Yaskawa INFORM job: A_ROOF_UPPER_0614_2_PAINT_62.JBI

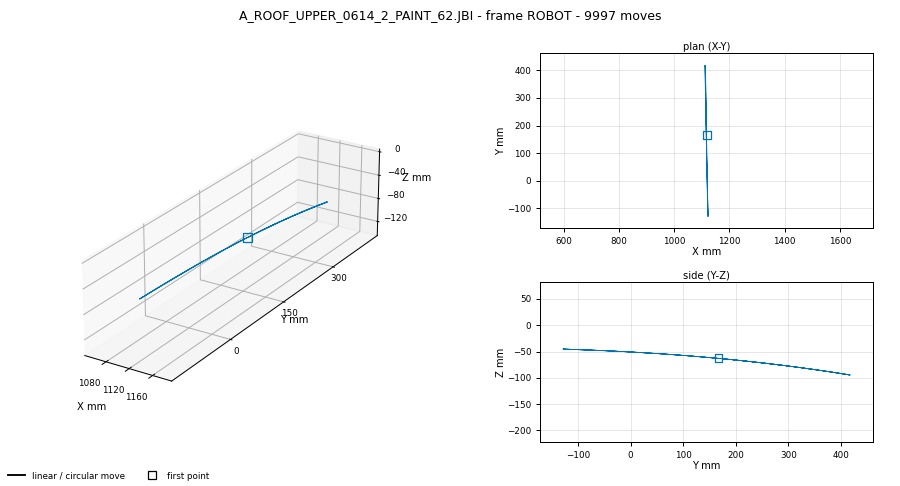
[picture p0: tool path of A_ROOF_UPPER_0614_2_PAINT_62.JBI in frame ROBOT, 9997 of 9997 moves have a stored position in this frame; points joined in program order, loops and branches not executed]
/JOB
//NAME A_ROOF_UPPER_0614_2_PAINT62
//POS
///NPOS 9997,0,0,0,0,0
///TOOL 1
///USER 0
///POSTYPE ROBOT
///RECTAN
///RCONF 1,0,0,0,0,0,0,0,0,0,0,0,0,0,0,0,0,0,0,0,0,0,0,0
C00000=1117.726,167.030,-62.893,-179.337,8.959,149.560
C00001=1117.722,167.279,-62.915,-179.335,8.962,149.560
C00002=1117.717,167.528,-62.939,-179.333,8.966,149.560
C00003=1117.713,167.777,-62.962,-179.330,8.969,149.560
C00004=1117.708,168.025,-62.984,-179.328,8.972,149.560
C00005=1117.703,168.274,-63.008,-179.326,8.975,149.560
C00006=1117.699,168.523,-63.031,-179.324,8.978,149.560
C00007=1117.695,168.772,-63.054,-179.321,8.981,149.560
C00008=1117.690,169.021,-63.077,-179.319,8.985,149.561
C00009=1117.685,169.270,-63.101,-179.317,8.988,149.561
C00010=1117.681,169.519,-63.124,-179.315,8.990,149.561
C00011=1117.676,169.767,-63.146,-179.313,8.993,149.561
C00012=1117.671,170.016,-63.170,-179.310,8.997,149.561
C00013=1117.667,170.265,-63.193,-179.308,9.000,149.561
C00014=1117.662,170.514,-63.217,-179.306,9.002,149.561
C00015=1117.658,170.763,-63.239,-179.304,9.005,149.561
C00016=1117.653,170.977,-63.260,-179.302,9.008,149.561
C00017=1117.650,171.190,-63.279,-179.300,9.010,149.561
C00018=1117.646,171.404,-63.299,-179.298,9.014,149.562
C00019=1117.642,171.619,-63.319,-179.296,9.016,149.562
C00020=1117.638,171.833,-63.339,-179.294,9.018,149.562
C00021=1117.634,172.046,-63.359,-179.292,9.021,149.562
C00022=1117.630,172.260,-63.379,-179.291,9.023,149.562
C00023=1117.626,172.474,-63.399,-179.288,9.026,149.562
C00024=1117.621,172.723,-63.422,-179.286,9.029,149.562
C00025=1117.617,172.971,-63.446,-179.284,9.032,149.562
C00026=1117.613,173.220,-63.469,-179.282,9.035,149.562
C00027=1117.608,173.469,-63.493,-179.280,9.038,149.562
C00028=1117.603,173.718,-63.516,-179.278,9.041,149.562
C00029=1117.599,173.967,-63.539,-179.275,9.044,149.562
C00030=1117.594,174.216,-63.563,-179.273,9.047,149.563
C00031=1117.590,174.464,-63.587,-179.271,9.050,149.563
C00032=1117.585,174.713,-63.610,-179.269,9.053,149.563
C00033=1117.581,174.962,-63.633,-179.267,9.056,149.563
C00034=1117.576,175.211,-63.656,-179.264,9.059,149.563
C00035=1117.572,175.460,-63.680,-179.262,9.062,149.563
C00036=1117.567,175.709,-63.704,-179.260,9.064,149.563
C00037=1117.562,175.958,-63.727,-179.258,9.068,149.563
C00038=1117.558,176.207,-63.750,-179.256,9.071,149.563
C00039=1117.553,176.455,-63.775,-179.254,9.073,149.563
C00040=1117.549,176.704,-63.798,-179.251,9.076,149.564
C00041=1117.544,176.953,-63.821,-179.249,9.080,149.564
C00042=1117.540,177.202,-63.845,-179.247,9.082,149.564
C00043=1117.535,177.451,-63.869,-179.245,9.085,149.564
C00044=1117.530,177.700,-63.892,-179.242,9.089,149.564
C00045=1117.526,177.948,-63.916,-179.241,9.091,149.564
C00046=1117.521,178.197,-63.939,-179.238,9.094,149.564
C00047=1117.517,178.445,-63.964,-179.236,9.098,149.564
C00048=1117.512,178.694,-63.987,-179.234,9.100,149.564
C00049=1117.507,178.943,-64.010,-179.232,9.103,149.564
C00050=1117.503,179.192,-64.034,-179.230,9.106,149.565
C00051=1117.499,179.442,-64.058,-179.228,9.109,149.565
C00052=1117.494,179.690,-64.082,-179.224,9.113,149.565
C00053=1117.490,179.939,-64.106,-179.222,9.116,149.565
C00054=1117.485,180.187,-64.130,-179.219,9.119,149.565
C00055=1117.481,180.437,-64.153,-179.217,9.122,149.565
C00056=1117.476,180.685,-64.177,-179.214,9.125,149.565
C00057=1117.471,180.934,-64.200,-179.211,9.128,149.565
C00058=1117.467,181.182,-64.224,-179.209,9.131,149.565
C00059=1117.462,181.432,-64.248,-179.206,9.134,149.565
C00060=1117.458,181.681,-64.273,-179.204,9.137,149.565
C00061=1117.453,181.930,-64.296,-179.201,9.141,149.565
C00062=1117.449,182.178,-64.320,-179.199,9.144,149.565
C00063=1117.444,182.427,-64.344,-179.196,9.147,149.565
C00064=1117.440,182.676,-64.368,-179.194,9.150,149.565
C00065=1117.435,182.924,-64.392,-179.191,9.153,149.565
C00066=1117.430,183.173,-64.416,-179.189,9.156,149.565
C00067=1117.426,183.423,-64.440,-179.186,9.159,149.565
C00068=1117.422,183.671,-64.464,-179.183,9.162,149.565
C00069=1117.417,183.920,-64.488,-179.181,9.165,149.565
C00070=1117.413,184.168,-64.512,-179.178,9.168,149.565
C00071=1117.407,184.417,-64.536,-179.176,9.171,149.565
C00072=1117.404,184.631,-64.557,-179.174,9.174,149.565
C00073=1117.400,184.845,-64.578,-179.172,9.176,149.565
C00074=1117.396,185.059,-64.598,-179.170,9.178,149.565
C00075=1117.393,185.272,-64.619,-179.167,9.181,149.565
C00076=1117.388,185.485,-64.640,-179.166,9.184,149.565
C00077=1117.384,185.699,-64.660,-179.164,9.186,149.565
C00078=1117.381,185.913,-64.681,-179.162,9.188,149.565
C00079=1117.377,186.127,-64.702,-179.159,9.191,149.566
C00080=1117.372,186.375,-64.726,-179.157,9.194,149.566
C00081=1117.368,186.624,-64.750,-179.154,9.197,149.565
C00082=1117.363,186.873,-64.775,-179.152,9.200,149.565
C00083=1117.359,187.122,-64.799,-179.150,9.202,149.565
C00084=1117.354,187.371,-64.822,-179.147,9.205,149.566
C00085=1117.350,187.620,-64.847,-179.145,9.208,149.566
C00086=1117.345,187.868,-64.871,-179.143,9.211,149.566
C00087=1117.341,188.117,-64.896,-179.140,9.214,149.566
C00088=1117.336,188.366,-64.920,-179.138,9.217,149.566
C00089=1117.332,188.615,-64.945,-179.136,9.219,149.566
C00090=1117.327,188.863,-64.969,-179.134,9.222,149.566
C00091=1117.322,189.112,-64.993,-179.131,9.225,149.566
C00092=1117.318,189.360,-65.017,-179.129,9.228,149.566
C00093=1117.313,189.610,-65.042,-179.127,9.231,149.566
C00094=1117.309,189.858,-65.067,-179.125,9.233,149.566
C00095=1117.305,190.106,-65.091,-179.122,9.236,149.566
C00096=1117.300,190.356,-65.115,-179.120,9.239,149.566
C00097=1117.295,190.605,-65.139,-179.118,9.242,149.566
C00098=1117.291,190.853,-65.164,-179.116,9.244,149.566
C00099=1117.287,191.102,-65.189,-179.114,9.247,149.566
C00100=1117.282,191.351,-65.214,-179.112,9.250,149.566
C00101=1117.277,191.599,-65.238,-179.109,9.253,149.566
C00102=1117.273,191.849,-65.263,-179.107,9.255,149.566
C00103=1117.268,192.097,-65.287,-179.105,9.258,149.567
C00104=1117.264,192.345,-65.311,-179.103,9.261,149.567
C00105=1117.259,192.595,-65.336,-179.101,9.263,149.567
C00106=1117.255,192.843,-65.360,-179.099,9.266,149.567
C00107=1117.250,193.092,-65.385,-179.097,9.269,149.567
C00108=1117.246,193.341,-65.409,-179.095,9.272,149.567
C00109=1117.241,193.590,-65.434,-179.093,9.274,149.567
C00110=1117.237,193.838,-65.458,-179.091,9.277,149.567
C00111=1117.232,194.087,-65.483,-179.089,9.280,149.567
C00112=1117.228,194.336,-65.508,-179.087,9.282,149.567
C00113=1117.223,194.585,-65.533,-179.085,9.285,149.568
C00114=1117.218,194.834,-65.557,-179.083,9.288,149.568
C00115=1117.214,195.082,-65.581,-179.081,9.291,149.568
C00116=1117.210,195.331,-65.607,-179.080,9.293,149.568
C00117=1117.205,195.579,-65.631,-179.077,9.296,149.568
C00118=1117.201,195.829,-65.656,-179.076,9.299,149.568
C00119=1117.196,196.077,-65.680,-179.074,9.301,149.568
C00120=1117.192,196.325,-65.706,-179.072,9.305,149.568
C00121=1117.187,196.575,-65.731,-179.069,9.308,149.568
C00122=1117.183,196.823,-65.755,-179.066,9.311,149.568
C00123=1117.178,197.073,-65.780,-179.063,9.315,149.568
C00124=1117.174,197.320,-65.805,-179.059,9.318,149.568
C00125=1117.169,197.570,-65.830,-179.057,9.321,149.568
C00126=1117.164,197.818,-65.854,-179.053,9.325,149.568
C00127=1117.161,198.067,-65.879,-179.051,9.328,149.568
C00128=1117.157,198.280,-65.901,-179.048,9.331,149.568
C00129=1117.153,198.494,-65.922,-179.045,9.334,149.568
C00130=1117.149,198.707,-65.943,-179.043,9.336,149.568
C00131=1117.145,198.921,-65.965,-179.040,9.339,149.568
C00132=1117.141,199.135,-65.986,-179.037,9.341,149.568
C00133=1117.138,199.348,-66.008,-179.035,9.345,149.568
C00134=1117.133,199.561,-66.029,-179.033,9.347,149.568
C00135=1117.130,199.775,-66.051,-179.030,9.350,149.568
C00136=1117.125,200.025,-66.076,-179.027,9.352,149.568
C00137=1117.121,200.273,-66.101,-179.024,9.356,149.568
C00138=1117.116,200.522,-66.126,-179.021,9.359,149.568
C00139=1117.112,200.770,-66.151,-179.018,9.362,149.567
C00140=1117.107,201.019,-66.176,-179.014,9.365,149.567
C00141=1117.103,201.267,-66.201,-179.012,9.368,149.567
C00142=1117.098,201.517,-66.226,-179.009,9.371,149.567
C00143=1117.094,201.765,-66.251,-179.006,9.374,149.567
C00144=1117.090,202.013,-66.277,-179.003,9.377,149.567
C00145=1117.085,202.262,-66.301,-179.000,9.381,149.567
C00146=1117.080,202.511,-66.327,-178.997,9.383,149.567
C00147=1117.076,202.760,-66.352,-178.994,9.386,149.567
C00148=1117.072,203.008,-66.377,-178.991,9.389,149.567
C00149=1117.068,203.257,-66.403,-178.988,9.391,149.566
C00150=1117.062,203.506,-66.427,-178.986,9.395,149.566
C00151=1117.058,203.755,-66.453,-178.982,9.398,149.566
C00152=1117.054,204.003,-66.479,-178.979,9.401,149.566
C00153=1117.049,204.251,-66.504,-178.976,9.404,149.566
C00154=1117.045,204.501,-66.529,-178.974,9.407,149.566
C00155=1117.040,204.749,-66.555,-178.971,9.409,149.566
C00156=1117.036,204.997,-66.580,-178.968,9.412,149.566
C00157=1117.032,205.246,-66.606,-178.965,9.415,149.566
C00158=1117.027,205.495,-66.630,-178.962,9.418,149.566
C00159=1117.023,205.744,-66.656,-178.959,9.421,149.566
C00160=1117.018,205.993,-66.682,-178.956,9.424,149.565
C00161=1117.014,206.241,-66.707,-178.954,9.427,149.566
C00162=1117.009,206.489,-66.733,-178.951,9.429,149.565
C00163=1117.004,206.738,-66.758,-178.948,9.432,149.565
C00164=1117.000,206.987,-66.783,-178.945,9.435,149.565
C00165=1116.996,207.236,-66.809,-178.942,9.438,149.565
C00166=1116.992,207.485,-66.835,-178.939,9.441,149.565
C00167=1116.987,207.733,-66.860,-178.937,9.444,149.565
C00168=1116.983,207.982,-66.886,-178.934,9.447,149.565
C00169=1116.978,208.230,-66.912,-178.931,9.449,149.565
C00170=1116.973,208.478,-66.937,-178.929,9.452,149.565
C00171=1116.969,208.727,-66.963,-178.926,9.455,149.565
C00172=1116.965,208.976,-66.989,-178.923,9.458,149.565
C00173=1116.960,209.224,-67.014,-178.920,9.461,149.565
C00174=1116.956,209.473,-67.040,-178.918,9.464,149.565
C00175=1116.951,209.722,-67.066,-178.915,9.467,149.565
C00176=1116.947,209.971,-67.092,-178.912,9.470,149.565
C00177=1116.942,210.219,-67.117,-178.909,9.473,149.564
C00178=1116.938,210.468,-67.143,-178.907,9.476,149.565
C00179=1116.934,210.717,-67.169,-178.905,9.478,149.565
C00180=1116.929,210.965,-67.195,-178.902,9.481,149.564
C00181=1116.924,211.213,-67.220,-178.899,9.484,149.564
C00182=1116.920,211.462,-67.246,-178.897,9.487,149.565
C00183=1116.916,211.711,-67.271,-178.894,9.490,149.564
C00184=1116.912,211.925,-67.294,-178.892,9.492,149.564
C00185=1116.908,212.137,-67.316,-178.889,9.495,149.564
C00186=1116.904,212.351,-67.339,-178.887,9.498,149.565
C00187=1116.900,212.565,-67.360,-178.885,9.501,149.565
C00188=1116.896,212.779,-67.383,-178.883,9.503,149.565
C00189=1116.893,212.992,-67.405,-178.881,9.505,149.565
C00190=1116.889,213.205,-67.427,-178.879,9.509,149.565
C00191=1116.885,213.418,-67.450,-178.877,9.511,149.565
C00192=1116.881,213.667,-67.476,-178.875,9.513,149.565
C00193=1116.877,213.916,-67.501,-178.872,9.516,149.565
C00194=1116.872,214.165,-67.527,-178.870,9.519,149.565
C00195=1116.868,214.413,-67.554,-178.868,9.522,149.565
C00196=1116.863,214.661,-67.580,-178.866,9.525,149.565
C00197=1116.859,214.910,-67.605,-178.864,9.528,149.565
C00198=1116.855,215.159,-67.631,-178.862,9.531,149.566
C00199=1116.850,215.407,-67.658,-178.860,9.533,149.566
C00200=1116.846,215.656,-67.684,-178.857,9.536,149.566
C00201=1116.841,215.905,-67.710,-178.856,9.539,149.566
C00202=1116.837,216.153,-67.737,-178.853,9.542,149.566
C00203=1116.832,216.402,-67.762,-178.851,9.545,149.566
C00204=1116.828,216.650,-67.788,-178.849,9.548,149.566
C00205=1116.824,216.899,-67.814,-178.847,9.551,149.566
C00206=1116.819,217.148,-67.841,-178.844,9.554,149.566
C00207=1116.815,217.396,-67.866,-178.842,9.557,149.567
C00208=1116.811,217.645,-67.893,-178.840,9.560,149.567
C00209=1116.806,217.894,-67.919,-178.838,9.563,149.567
C00210=1116.802,218.142,-67.946,-178.835,9.566,149.567
C00211=1116.798,218.391,-67.971,-178.833,9.569,149.567
C00212=1116.793,218.639,-67.999,-178.831,9.572,149.567
C00213=1116.788,218.887,-68.024,-178.829,9.575,149.567
C00214=1116.784,219.136,-68.050,-178.826,9.578,149.567
C00215=1116.779,219.385,-68.077,-178.824,9.581,149.567
C00216=1116.775,219.633,-68.103,-178.821,9.585,149.567
C00217=1116.770,219.882,-68.130,-178.819,9.588,149.568
C00218=1116.766,220.130,-68.156,-178.817,9.591,149.568
C00219=1116.762,220.379,-68.182,-178.814,9.594,149.568
C00220=1116.758,220.627,-68.209,-178.812,9.597,149.568
C00221=1116.753,220.876,-68.235,-178.810,9.600,149.568
C00222=1116.749,221.125,-68.262,-178.807,9.603,149.568
C00223=1116.744,221.374,-68.287,-178.805,9.606,149.568
C00224=1116.740,221.622,-68.314,-178.802,9.609,149.568
C00225=1116.736,221.870,-68.341,-178.800,9.612,149.568
C00226=1116.731,222.119,-68.367,-178.797,9.615,149.568
C00227=1116.727,222.368,-68.394,-178.794,9.618,149.568
C00228=1116.722,222.616,-68.421,-178.792,9.621,149.568
C00229=1116.718,222.865,-68.447,-178.789,9.625,149.569
C00230=1116.713,223.113,-68.474,-178.787,9.628,149.569
C00231=1116.710,223.362,-68.500,-178.784,9.632,149.569
C00232=1116.705,223.611,-68.526,-178.781,9.635,149.569
C00233=1116.701,223.859,-68.553,-178.779,9.638,149.569
C00234=1116.696,224.107,-68.580,-178.776,9.641,149.569
C00235=1116.692,224.356,-68.606,-178.774,9.644,149.569
C00236=1116.687,224.605,-68.633,-178.771,9.647,149.569
C00237=1116.683,224.853,-68.659,-178.768,9.650,149.569
C00238=1116.679,225.101,-68.686,-178.766,9.653,149.569
C00239=1116.674,225.350,-68.713,-178.762,9.657,149.569
C00240=1116.671,225.563,-68.736,-178.761,9.659,149.569
C00241=1116.667,225.777,-68.758,-178.758,9.662,149.569
C00242=1116.663,225.990,-68.782,-178.756,9.664,149.569
C00243=1116.659,226.203,-68.805,-178.753,9.667,149.569
C00244=1116.655,226.416,-68.828,-178.751,9.671,149.569
C00245=1116.652,226.630,-68.850,-178.748,9.672,149.569
C00246=1116.648,226.843,-68.874,-178.746,9.676,149.569
C00247=1116.644,227.056,-68.897,-178.744,9.678,149.569
C00248=1116.639,227.305,-68.924,-178.740,9.681,149.569
C00249=1116.635,227.553,-68.950,-178.738,9.685,149.569
C00250=1116.631,227.802,-68.977,-178.735,9.687,149.569
C00251=1116.627,228.051,-69.005,-178.732,9.690,149.569
C00252=1116.623,228.299,-69.031,-178.729,9.694,149.569
C00253=1116.618,228.548,-69.058,-178.726,9.697,149.569
C00254=1116.613,228.796,-69.085,-178.723,9.700,149.569
C00255=1116.609,229.044,-69.112,-178.720,9.703,149.569
C00256=1116.605,229.293,-69.139,-178.717,9.706,149.569
C00257=1116.600,229.541,-69.166,-178.714,9.709,149.569
C00258=1116.596,229.790,-69.193,-178.711,9.713,149.569
C00259=1116.592,230.039,-69.220,-178.708,9.715,149.568
C00260=1116.588,230.287,-69.247,-178.705,9.718,149.568
C00261=1116.583,230.536,-69.274,-178.702,9.722,149.568
C00262=1116.578,230.784,-69.301,-178.699,9.725,149.568
C00263=1116.574,231.033,-69.328,-178.696,9.728,149.568
C00264=1116.570,231.281,-69.356,-178.693,9.730,149.568
C00265=1116.566,231.529,-69.383,-178.690,9.733,149.568
C00266=1116.561,231.778,-69.410,-178.687,9.737,149.568
C00267=1116.557,232.026,-69.437,-178.684,9.740,149.568
C00268=1116.553,232.276,-69.464,-178.681,9.742,149.568
C00269=1116.548,232.524,-69.491,-178.678,9.745,149.568
C00270=1116.544,232.772,-69.519,-178.675,9.748,149.567
C00271=1116.539,233.020,-69.546,-178.672,9.751,149.567
C00272=1116.535,233.269,-69.572,-178.669,9.753,149.567
C00273=1116.531,233.518,-69.600,-178.666,9.757,149.567
C00274=1116.527,233.766,-69.628,-178.664,9.759,149.567
C00275=1116.522,234.014,-69.655,-178.661,9.762,149.567
C00276=1116.517,234.263,-69.682,-178.658,9.765,149.567
C00277=1116.514,234.511,-69.710,-178.655,9.768,149.567
C00278=1116.509,234.760,-69.737,-178.652,9.770,149.567
C00279=1116.504,235.008,-69.764,-178.649,9.773,149.567
C00280=1116.500,235.257,-69.792,-178.646,9.776,149.567
C00281=1116.496,235.505,-69.819,-178.644,9.778,149.566
C00282=1116.491,235.753,-69.847,-178.641,9.781,149.566
C00283=1116.487,236.002,-69.874,-178.638,9.784,149.566
C00284=1116.483,236.251,-69.902,-178.635,9.786,149.566
C00285=1116.478,236.499,-69.929,-178.632,9.789,149.566
C00286=1116.474,236.747,-69.956,-178.630,9.791,149.566
C00287=1116.470,236.996,-69.984,-178.627,9.794,149.566
C00288=1116.465,237.244,-70.012,-178.624,9.797,149.566
C00289=1116.461,237.492,-70.039,-178.622,9.799,149.566
C00290=1116.457,237.741,-70.067,-178.619,9.802,149.566
C00291=1116.453,237.989,-70.095,-178.617,9.805,149.566
C00292=1116.448,238.238,-70.122,-178.614,9.807,149.565
C00293=1116.444,238.486,-70.150,-178.611,9.810,149.565
C00294=1116.440,238.735,-70.177,-178.608,9.812,149.565
C00295=1116.436,238.983,-70.205,-178.606,9.815,149.565
C00296=1116.432,239.196,-70.228,-178.604,9.817,149.565
C00297=1116.428,239.410,-70.253,-178.601,9.819,149.565
C00298=1116.424,239.623,-70.276,-178.599,9.822,149.565
C00299=1116.420,239.836,-70.300,-178.597,9.824,149.565
C00300=1116.417,240.049,-70.323,-178.595,9.826,149.565
C00301=1116.413,240.263,-70.347,-178.593,9.828,149.565
C00302=1116.409,240.476,-70.371,-178.591,9.830,149.565
C00303=1116.405,240.688,-70.395,-178.589,9.832,149.565
C00304=1116.401,240.937,-70.423,-178.586,9.834,149.565
C00305=1116.397,241.185,-70.450,-178.584,9.837,149.565
C00306=1116.393,241.434,-70.479,-178.581,9.839,149.565
C00307=1116.389,241.682,-70.506,-178.579,9.842,149.565
C00308=1116.383,241.931,-70.534,-178.577,9.844,149.564
C00309=1116.380,242.179,-70.562,-178.574,9.848,149.565
C00310=1116.375,242.428,-70.589,-178.572,9.849,149.564
C00311=1116.371,242.676,-70.617,-178.570,9.852,149.564
C00312=1116.367,242.924,-70.645,-178.567,9.855,149.565
C00313=1116.362,243.173,-70.674,-178.565,9.857,149.564
C00314=1116.358,243.421,-70.701,-178.563,9.860,149.565
C00315=1116.353,243.669,-70.729,-178.560,9.862,149.564
C00316=1116.350,243.918,-70.757,-178.558,9.864,149.564
C00317=1116.345,244.166,-70.785,-178.556,9.867,149.565
C00318=1116.341,244.415,-70.813,-178.554,9.870,149.565
C00319=1116.336,244.663,-70.840,-178.552,9.872,149.564
C00320=1116.332,244.912,-70.869,-178.549,9.875,149.565
C00321=1116.327,245.160,-70.897,-178.547,9.877,149.565
C00322=1116.324,245.409,-70.925,-178.545,9.880,149.565
C00323=1116.319,245.656,-70.953,-178.543,9.882,149.565
C00324=1116.315,245.905,-70.981,-178.541,9.885,149.565
C00325=1116.310,246.153,-71.009,-178.539,9.887,149.565
C00326=1116.307,246.402,-71.038,-178.537,9.890,149.565
C00327=1116.302,246.650,-71.065,-178.535,9.892,149.565
C00328=1116.298,246.899,-71.093,-178.533,9.895,149.565
C00329=1116.293,247.147,-71.121,-178.531,9.897,149.565
C00330=1116.289,247.396,-71.149,-178.529,9.900,149.565
C00331=1116.284,247.644,-71.178,-178.525,9.903,149.565
C00332=1116.281,247.892,-71.206,-178.521,9.908,149.565
C00333=1116.276,248.140,-71.234,-178.516,9.912,149.565
C00334=1116.272,248.389,-71.262,-178.512,9.915,149.564
C00335=1116.267,248.637,-71.290,-178.508,9.919,149.564
C00336=1116.263,248.886,-71.319,-178.503,9.923,149.564
C00337=1116.259,249.134,-71.347,-178.500,9.926,149.564
C00338=1116.255,249.382,-71.375,-178.496,9.929,149.563
C00339=1116.251,249.631,-71.404,-178.492,9.932,149.563
C00340=1116.246,249.878,-71.432,-178.488,9.936,149.563
C00341=1116.242,250.127,-71.461,-178.484,9.939,149.563
C00342=1116.238,250.376,-71.489,-178.481,9.942,149.562
C00343=1116.233,250.624,-71.517,-178.477,9.945,149.562
C00344=1116.229,250.873,-71.545,-178.474,9.947,149.562
C00345=1116.224,251.120,-71.574,-178.470,9.951,149.562
C00346=1116.221,251.369,-71.603,-178.466,9.953,149.561
C00347=1116.216,251.618,-71.631,-178.463,9.956,149.561
C00348=1116.212,251.866,-71.659,-178.461,9.959,149.561
C00349=1116.208,252.114,-71.689,-178.457,9.961,149.561
C00350=1116.204,252.362,-71.717,-178.455,9.963,149.561
C00351=1116.199,252.611,-71.745,-178.452,9.966,149.561
C00352=1116.195,252.824,-71.770,-178.450,9.968,149.561
C00353=1116.192,253.036,-71.794,-178.447,9.970,149.560
C00354=1116.188,253.250,-71.819,-178.445,9.972,149.560
C00355=1116.185,253.463,-71.843,-178.444,9.973,149.560
C00356=1116.181,253.676,-71.868,-178.441,9.975,149.560
C00357=1116.178,253.889,-71.893,-178.439,9.977,149.560
C00358=1116.173,254.102,-71.917,-178.438,9.979,149.560
C00359=1116.169,254.315,-71.942,-178.436,9.981,149.560
C00360=1116.166,254.563,-71.971,-178.434,9.982,149.560
C00361=1116.161,254.812,-71.999,-178.432,9.985,149.560
C00362=1116.156,255.060,-72.028,-178.430,9.987,149.560
C00363=1116.153,255.308,-72.057,-178.429,9.988,149.560
C00364=1116.148,255.557,-72.085,-178.428,9.990,149.560
C00365=1116.144,255.805,-72.114,-178.426,9.992,149.560
C00366=1116.140,256.053,-72.143,-178.425,9.994,149.560
C00367=1116.136,256.302,-72.171,-178.422,9.997,149.560
C00368=1116.131,256.550,-72.200,-178.419,10.000,149.560
C00369=1116.127,256.798,-72.229,-178.416,10.003,149.560
C00370=1116.123,257.047,-72.258,-178.413,10.005,149.560
C00371=1116.118,257.295,-72.286,-178.411,10.008,149.560
C00372=1116.114,257.543,-72.315,-178.408,10.011,149.560
C00373=1116.110,257.792,-72.344,-178.405,10.014,149.560
C00374=1116.106,258.040,-72.373,-178.402,10.017,149.560
C00375=1116.101,258.288,-72.401,-178.399,10.019,149.560
C00376=1116.097,258.536,-72.431,-178.396,10.022,149.560
C00377=1116.093,258.784,-72.460,-178.393,10.025,149.560
C00378=1116.089,259.033,-72.488,-178.390,10.028,149.559
C00379=1116.085,259.281,-72.518,-178.388,10.031,149.560
C00380=1116.080,259.529,-72.546,-178.385,10.034,149.559
C00381=1116.076,259.778,-72.576,-178.382,10.036,149.559
C00382=1116.072,260.026,-72.605,-178.379,10.039,149.559
C00383=1116.068,260.275,-72.633,-178.376,10.042,149.559
C00384=1116.064,260.523,-72.663,-178.373,10.045,149.559
C00385=1116.059,260.770,-72.692,-178.370,10.047,149.559
C00386=1116.054,261.019,-72.720,-178.367,10.050,149.559
C00387=1116.050,261.268,-72.750,-178.364,10.053,149.559
C00388=1116.047,261.516,-72.779,-178.361,10.055,149.558
C00389=1116.042,261.764,-72.808,-178.357,10.059,149.558
C00390=1116.037,262.012,-72.837,-178.354,10.062,149.558
C00391=1116.033,262.260,-72.866,-178.352,10.064,149.558
C00392=1116.029,262.509,-72.896,-178.349,10.067,149.558
C00393=1116.025,262.757,-72.925,-178.345,10.069,149.558
C00394=1116.021,263.005,-72.954,-178.342,10.072,149.558
C00395=1116.016,263.254,-72.983,-178.339,10.076,149.558
C00396=1116.012,263.502,-73.013,-178.336,10.079,149.557
C00397=1116.008,263.749,-73.041,-178.332,10.081,149.557
C00398=1116.004,263.998,-73.071,-178.329,10.084,149.557
C00399=1116.000,264.246,-73.100,-178.325,10.087,149.557
C00400=1115.995,264.494,-73.129,-178.323,10.090,149.557
C00401=1115.991,264.743,-73.159,-178.320,10.092,149.556
C00402=1115.987,264.991,-73.188,-178.317,10.094,149.556
C00403=1115.983,265.239,-73.218,-178.314,10.097,149.556
C00404=1115.979,265.487,-73.247,-178.312,10.099,149.556
C00405=1115.975,265.736,-73.277,-178.309,10.102,149.556
C00406=1115.970,265.984,-73.306,-178.306,10.105,149.556
C00407=1115.966,266.232,-73.336,-178.304,10.107,149.556
C00408=1115.962,266.445,-73.360,-178.302,10.109,149.556
C00409=1115.958,266.658,-73.386,-178.299,10.111,149.556
C00410=1115.955,266.870,-73.411,-178.296,10.113,149.555
C00411=1115.951,267.084,-73.436,-178.294,10.115,149.555
C00412=1115.947,267.297,-73.462,-178.292,10.118,149.555
C00413=1115.944,267.509,-73.487,-178.290,10.120,149.555
C00414=1115.940,267.723,-73.512,-178.287,10.122,149.555
C00415=1115.937,267.936,-73.538,-178.285,10.124,149.555
C00416=1115.933,268.184,-73.568,-178.282,10.126,149.555
C00417=1115.928,268.432,-73.597,-178.279,10.129,149.555
C00418=1115.924,268.680,-73.626,-178.276,10.132,149.555
C00419=1115.920,268.929,-73.656,-178.274,10.134,149.555
C00420=1115.916,269.177,-73.685,-178.271,10.137,149.555
C00421=1115.911,269.425,-73.715,-178.268,10.139,149.554
C00422=1115.907,269.674,-73.745,-178.265,10.142,149.554
C00423=1115.903,269.921,-73.775,-178.263,10.144,149.554
C00424=1115.899,270.170,-73.805,-178.260,10.147,149.554
C00425=1115.895,270.418,-73.834,-178.257,10.150,149.554
C00426=1115.890,270.666,-73.863,-178.254,10.152,149.554
C00427=1115.886,270.914,-73.894,-178.251,10.155,149.554
C00428=1115.882,271.162,-73.924,-178.249,10.157,149.554
C00429=1115.877,271.411,-73.953,-178.246,10.160,149.554
C00430=1115.873,271.659,-73.983,-178.243,10.163,149.553
C00431=1115.869,271.907,-74.013,-178.240,10.165,149.553
C00432=1115.865,272.155,-74.042,-178.237,10.168,149.553
C00433=1115.860,272.403,-74.072,-178.234,10.171,149.553
C00434=1115.856,272.651,-74.102,-178.231,10.173,149.553
C00435=1115.852,272.899,-74.132,-178.229,10.175,149.553
C00436=1115.848,273.148,-74.161,-178.226,10.178,149.553
C00437=1115.843,273.396,-74.192,-178.223,10.181,149.553
C00438=1115.840,273.645,-74.222,-178.220,10.184,149.552
C00439=1115.836,273.892,-74.252,-178.217,10.186,149.552
C00440=1115.832,274.140,-74.282,-178.214,10.189,149.552
C00441=1115.827,274.389,-74.312,-178.211,10.192,149.552
C00442=1115.823,274.637,-74.342,-178.208,10.194,149.552
C00443=1115.819,274.885,-74.371,-178.205,10.197,149.552
C00444=1115.815,275.133,-74.401,-178.202,10.199,149.552
C00445=1115.810,275.381,-74.431,-178.199,10.202,149.552
C00446=1115.806,275.629,-74.462,-178.196,10.205,149.551
C00447=1115.802,275.878,-74.491,-178.194,10.207,149.551
C00448=1115.798,276.126,-74.522,-178.190,10.210,149.551
C00449=1115.794,276.374,-74.552,-178.187,10.213,149.551
C00450=1115.790,276.622,-74.582,-178.184,10.215,149.551
C00451=1115.785,276.870,-74.613,-178.181,10.218,149.551
C00452=1115.781,277.118,-74.642,-178.178,10.220,149.551
C00453=1115.777,277.367,-74.673,-178.175,10.223,149.550
C00454=1115.773,277.615,-74.703,-178.172,10.226,149.550
C00455=1115.769,277.862,-74.733,-178.169,10.229,149.550
C00456=1115.764,278.110,-74.763,-178.166,10.231,149.550
C00457=1115.760,278.359,-74.793,-178.163,10.234,149.550
C00458=1115.756,278.607,-74.824,-178.160,10.237,149.550
C00459=1115.752,278.855,-74.854,-178.157,10.239,149.549
C00460=1115.748,279.103,-74.884,-178.154,10.242,149.549
C00461=1115.743,279.351,-74.914,-178.151,10.245,149.549
C00462=1115.740,279.599,-74.945,-178.147,10.247,149.549
C00463=1115.736,279.847,-74.976,-178.145,10.250,149.549
C00464=1115.732,280.060,-75.001,-178.141,10.252,149.549
C00465=1115.728,280.273,-75.028,-178.139,10.254,149.548
C00466=1115.724,280.485,-75.054,-178.136,10.257,149.548
C00467=1115.721,280.698,-75.080,-178.134,10.259,149.548
C00468=1115.717,280.911,-75.106,-178.130,10.261,149.548
C00469=1115.714,281.124,-75.132,-178.128,10.263,149.548
C00470=1115.711,281.337,-75.158,-178.125,10.266,149.548
C00471=1115.707,281.550,-75.184,-178.123,10.268,149.548
C00472=1115.703,281.798,-75.215,-178.119,10.271,149.547
C00473=1115.698,282.046,-75.245,-178.116,10.273,149.547
C00474=1115.693,282.294,-75.275,-178.113,10.276,149.547
C00475=1115.690,282.543,-75.306,-178.110,10.278,149.547
C00476=1115.685,282.791,-75.337,-178.107,10.281,149.547
C00477=1115.682,283.038,-75.367,-178.104,10.284,149.547
C00478=1115.678,283.287,-75.398,-178.102,10.286,149.546
C00479=1115.673,283.535,-75.429,-178.098,10.288,149.546
C00480=1115.669,283.782,-75.459,-178.095,10.291,149.546
C00481=1115.665,284.031,-75.490,-178.092,10.293,149.546
C00482=1115.661,284.279,-75.520,-178.089,10.296,149.546
C00483=1115.657,284.527,-75.551,-178.086,10.299,149.546
C00484=1115.652,284.775,-75.582,-178.083,10.301,149.545
C00485=1115.649,285.023,-75.612,-178.080,10.304,149.545
C00486=1115.644,285.271,-75.643,-178.076,10.306,149.545
C00487=1115.640,285.520,-75.674,-178.074,10.308,149.545
C00488=1115.635,285.768,-75.705,-178.071,10.311,149.545
C00489=1115.632,286.015,-75.735,-178.068,10.314,149.544
C00490=1115.628,286.264,-75.766,-178.065,10.316,149.544
C00491=1115.623,286.511,-75.798,-178.062,10.319,149.544
C00492=1115.619,286.759,-75.828,-178.059,10.321,149.544
C00493=1115.615,287.008,-75.859,-178.055,10.324,149.544
C00494=1115.611,287.256,-75.890,-178.052,10.327,149.544
C00495=1115.607,287.504,-75.921,-178.050,10.328,149.543
C00496=1115.603,287.752,-75.951,-178.047,10.331,149.543
C00497=1115.599,287.999,-75.983,-178.044,10.334,149.543
C00498=1115.595,288.248,-76.014,-178.040,10.336,149.543
C00499=1115.590,288.496,-76.044,-178.038,10.339,149.543
C00500=1115.586,288.744,-76.076,-178.034,10.341,149.543
C00501=1115.582,288.992,-76.106,-178.031,10.344,149.542
C00502=1115.578,289.239,-76.137,-178.028,10.347,149.542
C00503=1115.574,289.488,-76.168,-178.025,10.349,149.542
C00504=1115.569,289.736,-76.199,-178.022,10.351,149.542
C00505=1115.565,289.984,-76.231,-178.019,10.354,149.542
C00506=1115.561,290.232,-76.261,-178.016,10.357,149.542
C00507=1115.557,290.480,-76.292,-178.013,10.359,149.541
C00508=1115.553,290.728,-76.324,-178.010,10.362,149.541
C00509=1115.549,290.976,-76.355,-178.007,10.364,149.541
C00510=1115.545,291.224,-76.386,-178.004,10.367,149.541
C00511=1115.541,291.472,-76.417,-178.001,10.369,149.541
C00512=1115.536,291.720,-76.448,-177.998,10.372,149.541
C00513=1115.533,291.968,-76.480,-177.994,10.375,149.540
C00514=1115.528,292.216,-76.511,-177.992,10.377,149.540
C00515=1115.525,292.464,-76.542,-177.989,10.379,149.540
C00516=1115.520,292.712,-76.573,-177.986,10.382,149.540
C00517=1115.517,292.960,-76.605,-177.983,10.384,149.540
C00518=1115.512,293.208,-76.635,-177.979,10.387,149.539
C00519=1115.508,293.456,-76.667,-177.977,10.390,149.539
C00520=1115.504,293.669,-76.694,-177.974,10.391,149.539
C00521=1115.501,293.882,-76.721,-177.971,10.394,149.539
C00522=1115.498,294.094,-76.748,-177.969,10.396,149.539
C00523=1115.494,294.307,-76.774,-177.966,10.398,149.539
C00524=1115.490,294.519,-76.801,-177.963,10.401,149.538
C00525=1115.486,294.732,-76.828,-177.961,10.402,149.538
C00526=1115.483,294.944,-76.855,-177.958,10.404,149.538
C00527=1115.480,295.158,-76.882,-177.955,10.407,149.538
C00528=1115.476,295.405,-76.913,-177.953,10.409,149.538
C00529=1115.472,295.653,-76.945,-177.950,10.412,149.538
C00530=1115.467,295.901,-76.976,-177.946,10.414,149.537
C00531=1115.464,296.149,-77.008,-177.943,10.417,149.537
C00532=1115.459,296.397,-77.039,-177.940,10.419,149.537
C00533=1115.455,296.645,-77.071,-177.937,10.422,149.537
C00534=1115.451,296.894,-77.103,-177.934,10.424,149.537
C00535=1115.447,297.141,-77.134,-177.931,10.427,149.537
C00536=1115.443,297.390,-77.166,-177.928,10.430,149.536
C00537=1115.438,297.637,-77.197,-177.925,10.432,149.536
C00538=1115.435,297.885,-77.229,-177.922,10.434,149.536
C00539=1115.431,298.133,-77.261,-177.919,10.437,149.536
C00540=1115.426,298.381,-77.291,-177.916,10.439,149.536
C00541=1115.422,298.629,-77.323,-177.913,10.442,149.536
C00542=1115.418,298.877,-77.356,-177.909,10.444,149.535
C00543=1115.414,299.125,-77.387,-177.907,10.447,149.535
C00544=1115.410,299.373,-77.419,-177.903,10.450,149.535
C00545=1115.406,299.621,-77.451,-177.900,10.452,149.535
C00546=1115.402,299.869,-77.482,-177.897,10.455,149.535
C00547=1115.398,300.117,-77.514,-177.894,10.458,149.535
C00548=1115.394,300.365,-77.546,-177.891,10.459,149.534
C00549=1115.389,300.612,-77.577,-177.888,10.462,149.534
C00550=1115.386,300.860,-77.609,-177.885,10.465,149.534
C00551=1115.382,301.109,-77.641,-177.882,10.467,149.534
C00552=1115.377,301.356,-77.673,-177.879,10.470,149.534
C00553=1115.373,301.604,-77.705,-177.876,10.472,149.534
C00554=1115.369,301.852,-77.737,-177.872,10.475,149.533
C00555=1115.364,302.100,-77.769,-177.870,10.478,149.533
C00556=1115.361,302.348,-77.801,-177.866,10.480,149.533
C00557=1115.357,302.596,-77.833,-177.863,10.483,149.533
C00558=1115.353,302.843,-77.864,-177.861,10.485,149.533
C00559=1115.348,303.092,-77.897,-177.858,10.487,149.532
C00560=1115.344,303.340,-77.928,-177.854,10.490,149.532
C00561=1115.341,303.588,-77.960,-177.851,10.493,149.532
C00562=1115.336,303.835,-77.992,-177.848,10.495,149.532
C00563=1115.332,304.083,-78.024,-177.845,10.498,149.532
C00564=1115.328,304.331,-78.056,-177.842,10.500,149.532
C00565=1115.324,304.580,-78.089,-177.839,10.503,149.531
C00566=1115.320,304.827,-78.121,-177.836,10.505,149.531
C00567=1115.315,305.075,-78.153,-177.833,10.508,149.531
C00568=1115.312,305.323,-78.185,-177.830,10.510,149.531
C00569=1115.308,305.571,-78.217,-177.827,10.512,149.531
C00570=1115.303,305.819,-78.249,-177.824,10.515,149.530
C00571=1115.300,306.066,-78.281,-177.820,10.517,149.530
C00572=1115.295,306.314,-78.314,-177.817,10.520,149.530
C00573=1115.291,306.562,-78.346,-177.814,10.523,149.530
C00574=1115.287,306.811,-78.378,-177.811,10.525,149.530
C00575=1115.283,307.057,-78.410,-177.808,10.528,149.530
C00576=1115.280,307.271,-78.438,-177.806,10.530,149.529
C00577=1115.276,307.483,-78.465,-177.803,10.532,149.529
C00578=1115.273,307.695,-78.493,-177.800,10.534,149.529
C00579=1115.269,307.908,-78.521,-177.798,10.536,149.529
C00580=1115.265,308.121,-78.548,-177.795,10.539,149.529
C00581=1115.262,308.333,-78.576,-177.792,10.541,149.529
C00582=1115.259,308.546,-78.604,-177.790,10.543,149.528
C00583=1115.255,308.758,-78.632,-177.787,10.545,149.528
C00584=1115.251,309.006,-78.664,-177.784,10.547,149.528
C00585=1115.247,309.254,-78.696,-177.781,10.550,149.528
C00586=1115.243,309.502,-78.729,-177.778,10.552,149.528
C00587=1115.239,309.749,-78.761,-177.774,10.555,149.528
C00588=1115.235,309.997,-78.794,-177.772,10.558,149.527
C00589=1115.231,310.245,-78.826,-177.768,10.560,149.527
C00590=1115.227,310.493,-78.859,-177.765,10.563,149.527
C00591=1115.222,310.741,-78.891,-177.762,10.565,149.527
C00592=1115.219,310.989,-78.924,-177.759,10.568,149.527
C00593=1115.215,311.237,-78.956,-177.756,10.570,149.527
C00594=1115.211,311.484,-78.989,-177.753,10.573,149.526
C00595=1115.207,311.733,-79.021,-177.750,10.575,149.526
C00596=1115.203,311.980,-79.055,-177.747,10.577,149.526
C00597=1115.198,312.228,-79.086,-177.744,10.580,149.526
C00598=1115.194,312.476,-79.119,-177.740,10.582,149.526
C00599=1115.190,312.723,-79.152,-177.738,10.585,149.526
C00600=1115.186,312.971,-79.184,-177.734,10.588,149.525
C00601=1115.182,313.219,-79.217,-177.731,10.590,149.525
C00602=1115.178,313.467,-79.250,-177.728,10.593,149.525
C00603=1115.174,313.715,-79.282,-177.725,10.595,149.525
C00604=1115.170,313.963,-79.316,-177.722,10.598,149.525
C00605=1115.166,314.211,-79.348,-177.719,10.600,149.524
C00606=1115.162,314.458,-79.381,-177.716,10.603,149.524
C00607=1115.158,314.706,-79.414,-177.713,10.605,149.524
C00608=1115.154,314.954,-79.446,-177.709,10.607,149.524
C00609=1115.150,315.202,-79.479,-177.707,10.610,149.524
C00610=1115.146,315.450,-79.512,-177.703,10.613,149.523
C00611=1115.142,315.697,-79.545,-177.700,10.615,149.523
C00612=1115.138,315.945,-79.578,-177.697,10.618,149.523
C00613=1115.134,316.193,-79.610,-177.694,10.620,149.523
C00614=1115.130,316.441,-79.643,-177.691,10.623,149.523
C00615=1115.126,316.688,-79.676,-177.687,10.625,149.523
C00616=1115.122,316.936,-79.709,-177.685,10.627,149.522
C00617=1115.118,317.184,-79.743,-177.682,10.630,149.522
C00618=1115.114,317.431,-79.775,-177.678,10.632,149.522
C00619=1115.110,317.680,-79.808,-177.675,10.635,149.522
C00620=1115.106,317.927,-79.841,-177.672,10.638,149.522
C00621=1115.102,318.175,-79.874,-177.669,10.640,149.522
C00622=1115.098,318.424,-79.907,-177.666,10.643,149.521
C00623=1115.095,318.671,-79.940,-177.663,10.645,149.521
C00624=1115.090,318.919,-79.973,-177.660,10.648,149.521
C00625=1115.086,319.166,-80.006,-177.656,10.650,149.521
C00626=1115.082,319.414,-80.039,-177.653,10.653,149.521
C00627=1115.078,319.662,-80.073,-177.651,10.655,149.520
C00628=1115.074,319.910,-80.106,-177.647,10.657,149.520
C00629=1115.070,320.157,-80.139,-177.644,10.660,149.520
C00630=1115.066,320.405,-80.172,-177.641,10.663,149.520
C00631=1115.062,320.653,-80.205,-177.638,10.665,149.520
C00632=1115.059,320.865,-80.234,-177.636,10.667,149.519
C00633=1115.056,321.078,-80.262,-177.633,10.670,149.519
C00634=1115.052,321.290,-80.290,-177.630,10.671,149.519
C00635=1115.049,321.503,-80.319,-177.627,10.674,149.519
C00636=1115.045,321.715,-80.347,-177.624,10.676,149.519
C00637=1115.042,321.927,-80.377,-177.622,10.678,149.519
C00638=1115.038,322.139,-80.405,-177.619,10.681,149.519
C00639=1115.035,322.352,-80.434,-177.616,10.682,149.518
C00640=1115.031,322.600,-80.467,-177.613,10.685,149.518
C00641=1115.027,322.847,-80.500,-177.610,10.688,149.518
C00642=1115.022,323.095,-80.533,-177.607,10.690,149.518
C00643=1115.019,323.343,-80.567,-177.604,10.693,149.518
C00644=1115.015,323.591,-80.600,-177.601,10.694,149.517
C00645=1115.011,323.838,-80.634,-177.598,10.697,149.517
C00646=1115.007,324.086,-80.667,-177.595,10.700,149.517
C00647=1115.003,324.334,-80.700,-177.592,10.702,149.517
C00648=1114.999,324.581,-80.734,-177.588,10.705,149.517
C00649=1114.995,324.829,-80.767,-177.585,10.707,149.517
C00650=1114.991,325.077,-80.800,-177.582,10.710,149.516
C00651=1114.987,325.324,-80.834,-177.579,10.712,149.516
C00652=1114.983,325.572,-80.867,-177.576,10.715,149.516
C00653=1114.980,325.820,-80.901,-177.572,10.717,149.516
C00654=1114.976,326.067,-80.935,-177.569,10.720,149.516
C00655=1114.972,326.315,-80.968,-177.566,10.723,149.515
C00656=1114.967,326.563,-81.002,-177.564,10.724,149.515
C00657=1114.964,326.811,-81.036,-177.560,10.727,149.515
C00658=1114.959,327.059,-81.069,-177.557,10.730,149.515
C00659=1114.956,327.306,-81.103,-177.554,10.732,149.515
C00660=1114.951,327.554,-81.136,-177.551,10.734,149.514
C00661=1114.948,327.801,-81.170,-177.548,10.737,149.514
C00662=1114.943,328.049,-81.204,-177.544,10.740,149.514
C00663=1114.939,328.297,-81.237,-177.541,10.742,149.514
C00664=1114.935,328.544,-81.271,-177.538,10.745,149.514
C00665=1114.932,328.793,-81.305,-177.535,10.747,149.514
C00666=1114.928,329.040,-81.339,-177.532,10.750,149.513
C00667=1114.923,329.287,-81.373,-177.529,10.752,149.513
C00668=1114.920,329.536,-81.407,-177.526,10.754,149.513
C00669=1114.916,329.783,-81.440,-177.523,10.757,149.513
C00670=1114.912,330.030,-81.474,-177.520,10.760,149.513
C00671=1114.907,330.278,-81.508,-177.516,10.762,149.512
C00672=1114.904,330.526,-81.542,-177.513,10.764,149.512
C00673=1114.900,330.773,-81.575,-177.510,10.767,149.512
C00674=1114.895,331.021,-81.610,-177.507,10.770,149.512
C00675=1114.892,331.269,-81.643,-177.503,10.772,149.512
C00676=1114.888,331.516,-81.677,-177.500,10.775,149.511
C00677=1114.884,331.763,-81.711,-177.497,10.777,149.511
C00678=1114.880,332.012,-81.745,-177.495,10.779,149.511
C00679=1114.876,332.259,-81.779,-177.491,10.781,149.511
C00680=1114.873,332.507,-81.813,-177.488,10.784,149.511
C00681=1114.868,332.755,-81.848,-177.485,10.787,149.511
C00682=1114.864,333.002,-81.881,-177.482,10.789,149.510
C00683=1114.860,333.250,-81.916,-177.478,10.792,149.510
C00684=1114.856,333.498,-81.950,-177.475,10.794,149.510
C00685=1114.853,333.745,-81.984,-177.472,10.797,149.510
C00686=1114.849,333.993,-82.018,-177.469,10.799,149.510
C00687=1114.844,334.240,-82.052,-177.466,10.802,149.510
C00688=1114.841,334.453,-82.081,-177.463,10.804,149.509
C00689=1114.838,334.665,-82.111,-177.461,10.806,149.509
C00690=1114.835,334.877,-82.140,-177.458,10.808,149.509
C00691=1114.831,335.089,-82.169,-177.455,10.810,149.509
C00692=1114.827,335.302,-82.199,-177.453,10.812,149.509
C00693=1114.824,335.514,-82.228,-177.450,10.815,149.509
C00694=1114.821,335.726,-82.258,-177.447,10.816,149.508
C00695=1114.817,335.938,-82.287,-177.444,10.819,149.508
C00696=1114.814,336.186,-82.320,-177.441,10.821,149.508
C00697=1114.810,336.433,-82.354,-177.438,10.823,149.508
C00698=1114.806,336.681,-82.389,-177.435,10.826,149.507
C00699=1114.802,336.929,-82.423,-177.432,10.828,149.507
C00700=1114.798,337.177,-82.458,-177.429,10.831,149.507
C00701=1114.794,337.424,-82.492,-177.425,10.833,149.507
C00702=1114.790,337.672,-82.527,-177.422,10.836,149.507
C00703=1114.786,337.919,-82.561,-177.419,10.839,149.507
C00704=1114.783,338.166,-82.596,-177.416,10.841,149.506
C00705=1114.778,338.414,-82.630,-177.412,10.844,149.506
C00706=1114.775,338.662,-82.665,-177.409,10.846,149.506
C00707=1114.770,338.909,-82.699,-177.407,10.848,149.506
C00708=1114.767,339.157,-82.733,-177.403,10.850,149.506
C00709=1114.763,339.404,-82.768,-177.400,10.853,149.505
C00710=1114.759,339.652,-82.803,-177.397,10.855,149.505
C00711=1114.755,339.900,-82.837,-177.393,10.858,149.505
C00712=1114.751,340.148,-82.871,-177.391,10.861,149.505
C00713=1114.747,340.394,-82.907,-177.387,10.863,149.505
C00714=1114.743,340.642,-82.941,-177.384,10.866,149.504
C00715=1114.739,340.890,-82.975,-177.381,10.868,149.504
C00716=1114.735,341.138,-83.010,-177.378,10.871,149.504
C00717=1114.731,341.385,-83.044,-177.374,10.873,149.504
C00718=1114.727,341.632,-83.080,-177.371,10.876,149.504
C00719=1114.723,341.880,-83.114,-177.368,10.877,149.503
C00720=1114.719,342.128,-83.148,-177.365,10.880,149.503
C00721=1114.716,342.376,-83.183,-177.362,10.883,149.503
C00722=1114.711,342.623,-83.218,-177.359,10.885,149.503
C00723=1114.708,342.870,-83.253,-177.356,10.888,149.503
C00724=1114.703,343.118,-83.287,-177.352,10.890,149.502
C00725=1114.700,343.365,-83.323,-177.349,10.892,149.502
C00726=1114.695,343.613,-83.357,-177.346,10.895,149.502
C00727=1114.692,343.860,-83.392,-177.343,10.898,149.502
C00728=1114.688,344.108,-83.427,-177.339,10.900,149.502
C00729=1114.684,344.355,-83.461,-177.336,10.903,149.501
C00730=1114.680,344.603,-83.497,-177.333,10.904,149.501
C00731=1114.676,344.851,-83.532,-177.330,10.907,149.501
C00732=1114.673,345.098,-83.566,-177.327,10.910,149.501
C00733=1114.669,345.346,-83.601,-177.324,10.912,149.501
C00734=1114.664,345.593,-83.636,-177.320,10.914,149.500
C00735=1114.660,345.841,-83.671,-177.317,10.917,149.500
C00736=1114.657,346.088,-83.707,-177.314,10.919,149.500
C00737=1114.652,346.336,-83.741,-177.311,10.922,149.500
C00738=1114.649,346.583,-83.776,-177.308,10.925,149.500
C00739=1114.645,346.831,-83.811,-177.304,10.927,149.499
C00740=1114.641,347.078,-83.846,-177.301,10.930,149.499
C00741=1114.637,347.326,-83.881,-177.298,10.932,149.499
C00742=1114.633,347.573,-83.916,-177.295,10.934,149.499
C00743=1114.629,347.820,-83.952,-177.292,10.936,149.499
C00744=1114.626,348.032,-83.981,-177.289,10.939,149.498
C00745=1114.623,348.245,-84.011,-177.287,10.941,149.498
C00746=1114.619,348.457,-84.042,-177.284,10.943,149.498
C00747=1114.616,348.669,-84.071,-177.281,10.945,149.498
C00748=1114.613,348.880,-84.102,-177.278,10.947,149.498
C00749=1114.609,349.093,-84.132,-177.276,10.949,149.498
C00750=1114.606,349.305,-84.162,-177.273,10.952,149.498
C00751=1114.603,349.517,-84.192,-177.270,10.953,149.497
C00752=1114.599,349.764,-84.227,-177.267,10.956,149.497
C00753=1114.596,350.012,-84.263,-177.263,10.958,149.497
C00754=1114.592,350.260,-84.298,-177.260,10.961,149.497
C00755=1114.587,350.507,-84.333,-177.256,10.964,149.496
C00756=1114.584,350.754,-84.368,-177.253,10.966,149.496
C00757=1114.580,351.002,-84.404,-177.249,10.969,149.496
C00758=1114.576,351.249,-84.439,-177.246,10.971,149.496
C00759=1114.572,351.497,-84.474,-177.243,10.974,149.496
C00760=1114.568,351.744,-84.509,-177.240,10.976,149.495
C00761=1114.564,351.992,-84.545,-177.236,10.979,149.495
C00762=1114.561,352.239,-84.581,-177.233,10.981,149.495
C00763=1114.557,352.487,-84.616,-177.229,10.983,149.494
C00764=1114.553,352.735,-84.652,-177.226,10.986,149.494
C00765=1114.548,352.981,-84.687,-177.223,10.988,149.494
C00766=1114.545,353.229,-84.723,-177.219,10.991,149.494
C00767=1114.541,353.476,-84.759,-177.216,10.993,149.494
C00768=1114.537,353.724,-84.794,-177.213,10.996,149.493
C00769=1114.534,353.971,-84.830,-177.209,10.998,149.493
C00770=1114.530,354.219,-84.865,-177.205,11.001,149.493
C00771=1114.526,354.466,-84.900,-177.202,11.004,149.493
C00772=1114.522,354.713,-84.936,-177.198,11.006,149.492
C00773=1114.519,354.961,-84.971,-177.195,11.008,149.492
C00774=1114.514,355.208,-85.008,-177.192,11.011,149.492
C00775=1114.510,355.456,-85.043,-177.188,11.013,149.492
C00776=1114.507,355.703,-85.079,-177.185,11.016,149.491
C00777=1114.503,355.951,-85.114,-177.182,11.018,149.491
C00778=1114.499,356.198,-85.149,-177.178,11.020,149.491
C00779=1114.495,356.445,-85.185,-177.175,11.023,149.491
C00780=1114.491,356.693,-85.221,-177.172,11.025,149.490
C00781=1114.487,356.941,-85.257,-177.168,11.028,149.490
C00782=1114.484,357.187,-85.293,-177.165,11.030,149.490
C00783=1114.480,357.435,-85.328,-177.162,11.033,149.490
C00784=1114.476,357.683,-85.365,-177.158,11.035,149.489
C00785=1114.472,357.930,-85.400,-177.155,11.037,149.489
C00786=1114.468,358.178,-85.436,-177.151,11.040,149.489
C00787=1114.465,358.425,-85.472,-177.148,11.042,149.489
C00788=1114.461,358.672,-85.508,-177.145,11.045,149.488
C00789=1114.457,358.920,-85.544,-177.141,11.047,149.488
C00790=1114.454,359.167,-85.580,-177.138,11.049,149.488
C00791=1114.450,359.414,-85.615,-177.134,11.052,149.488
C00792=1114.446,359.662,-85.652,-177.131,11.054,149.487
C00793=1114.442,359.909,-85.688,-177.128,11.057,149.487
C00794=1114.439,360.156,-85.723,-177.124,11.059,149.487
C00795=1114.434,360.404,-85.760,-177.121,11.061,149.487
C00796=1114.431,360.651,-85.796,-177.117,11.064,149.486
C00797=1114.427,360.899,-85.831,-177.114,11.066,149.486
C00798=1114.423,361.146,-85.868,-177.111,11.069,149.486
C00799=1114.419,361.393,-85.904,-177.107,11.071,149.485
C00800=1114.416,361.605,-85.935,-177.104,11.073,149.485
C00801=1114.413,361.817,-85.965,-177.102,11.075,149.485
C00802=1114.409,362.029,-85.996,-177.099,11.077,149.485
C00803=1114.406,362.241,-86.028,-177.096,11.079,149.485
C00804=1114.403,362.453,-86.059,-177.093,11.081,149.484
C00805=1114.400,362.664,-86.089,-177.090,11.083,149.484
C00806=1114.396,362.876,-86.120,-177.087,11.085,149.484
C00807=1114.393,363.089,-86.151,-177.084,11.087,149.484
C00808=1114.390,363.336,-86.188,-177.081,11.089,149.484
C00809=1114.386,363.583,-86.224,-177.078,11.092,149.483
C00810=1114.382,363.831,-86.260,-177.074,11.094,149.483
C00811=1114.379,364.078,-86.296,-177.071,11.097,149.483
C00812=1114.374,364.325,-86.332,-177.067,11.099,149.482
C00813=1114.371,364.572,-86.369,-177.064,11.102,149.482
C00814=1114.367,364.819,-86.406,-177.061,11.104,149.482
C00815=1114.363,365.067,-86.441,-177.057,11.106,149.482
C00816=1114.359,365.314,-86.478,-177.054,11.109,149.481
C00817=1114.356,365.561,-86.514,-177.050,11.111,149.481
C00818=1114.351,365.809,-86.550,-177.047,11.114,149.481
C00819=1114.348,366.057,-86.588,-177.044,11.116,149.481
C00820=1114.344,366.304,-86.624,-177.041,11.119,149.481
C00821=1114.340,366.551,-86.660,-177.037,11.120,149.480
C00822=1114.337,366.798,-86.696,-177.034,11.122,149.480
C00823=1114.333,367.045,-86.733,-177.031,11.125,149.480
C00824=1114.329,367.292,-86.769,-177.028,11.127,149.480
C00825=1114.325,367.539,-86.806,-177.024,11.130,149.479
C00826=1114.321,367.787,-86.842,-177.021,11.132,149.479
C00827=1114.318,368.035,-86.879,-177.017,11.134,149.479
C00828=1114.314,368.282,-86.916,-177.014,11.137,149.479
C00829=1114.310,368.529,-86.953,-177.011,11.139,149.478
C00830=1114.306,368.776,-86.989,-177.007,11.142,149.478
C00831=1114.302,369.023,-87.026,-177.004,11.144,149.478
C00832=1114.299,369.270,-87.062,-177.001,11.147,149.478
C00833=1114.295,369.519,-87.099,-176.997,11.149,149.477
C00834=1114.291,369.766,-87.135,-176.994,11.151,149.477
C00835=1114.288,370.013,-87.172,-176.990,11.154,149.477
C00836=1114.284,370.260,-87.209,-176.987,11.156,149.477
C00837=1114.280,370.507,-87.245,-176.984,11.159,149.476
C00838=1114.276,370.755,-87.283,-176.981,11.161,149.476
C00839=1114.273,371.002,-87.319,-176.977,11.164,149.476
C00840=1114.269,371.249,-87.356,-176.974,11.166,149.476
C00841=1114.265,371.496,-87.393,-176.971,11.169,149.476
C00842=1114.262,371.744,-87.429,-176.967,11.171,149.475
C00843=1114.258,371.991,-87.466,-176.964,11.174,149.475
C00844=1114.254,372.238,-87.503,-176.961,11.176,149.475
C00845=1114.250,372.485,-87.541,-176.957,11.178,149.475
C00846=1114.246,372.733,-87.578,-176.954,11.181,149.474
C00847=1114.243,372.980,-87.614,-176.950,11.183,149.474
C00848=1114.239,373.227,-87.651,-176.947,11.186,149.474
C00849=1114.235,373.474,-87.688,-176.944,11.188,149.474
C00850=1114.231,373.722,-87.725,-176.941,11.191,149.474
C00851=1114.227,373.969,-87.762,-176.937,11.193,149.473
C00852=1114.224,374.215,-87.799,-176.934,11.196,149.473
C00853=1114.221,374.463,-87.836,-176.931,11.198,149.473
C00854=1114.217,374.710,-87.873,-176.928,11.200,149.473
C00855=1114.212,374.958,-87.910,-176.925,11.202,149.473
C00856=1114.210,375.170,-87.942,-176.922,11.205,149.473
C00857=1114.206,375.381,-87.973,-176.919,11.207,149.472
C00858=1114.203,375.592,-88.005,-176.916,11.209,149.472
C00859=1114.200,375.804,-88.037,-176.914,11.211,149.472
C00860=1114.196,376.016,-88.069,-176.910,11.214,149.472
C00861=1114.194,376.228,-88.101,-176.908,11.216,149.472
C00862=1114.190,376.439,-88.133,-176.905,11.218,149.472
C00863=1114.187,376.652,-88.164,-176.902,11.220,149.471
C00864=1114.183,376.899,-88.202,-176.899,11.223,149.471
C00865=1114.179,377.146,-88.239,-176.896,11.225,149.471
C00866=1114.176,377.393,-88.276,-176.893,11.228,149.471
C00867=1114.172,377.640,-88.313,-176.889,11.230,149.471
C00868=1114.168,377.888,-88.351,-176.886,11.233,149.471
C00869=1114.165,378.135,-88.388,-176.883,11.235,149.470
C00870=1114.161,378.382,-88.425,-176.879,11.238,149.470
C00871=1114.157,378.629,-88.463,-176.877,11.241,149.470
C00872=1114.153,378.876,-88.500,-176.873,11.243,149.470
C00873=1114.150,379.123,-88.537,-176.870,11.246,149.470
C00874=1114.146,379.371,-88.575,-176.867,11.248,149.470
C00875=1114.142,379.617,-88.612,-176.864,11.251,149.470
C00876=1114.139,379.865,-88.649,-176.860,11.253,149.469
C00877=1114.135,380.112,-88.687,-176.857,11.256,149.469
C00878=1114.131,380.360,-88.724,-176.854,11.258,149.469
C00879=1114.128,380.606,-88.762,-176.851,11.261,149.469
C00880=1114.124,380.853,-88.799,-176.848,11.264,149.469
C00881=1114.120,381.101,-88.837,-176.844,11.266,149.469
C00882=1114.117,381.347,-88.874,-176.841,11.269,149.469
C00883=1114.113,381.595,-88.911,-176.838,11.271,149.468
C00884=1114.109,381.842,-88.949,-176.835,11.274,149.468
C00885=1114.105,382.089,-88.987,-176.832,11.277,149.468
C00886=1114.101,382.336,-89.024,-176.829,11.279,149.468
C00887=1114.098,382.584,-89.062,-176.825,11.283,149.468
C00888=1114.094,382.830,-89.100,-176.822,11.285,149.468
C00889=1114.091,383.078,-89.138,-176.819,11.288,149.468
C00890=1114.087,383.325,-89.175,-176.816,11.291,149.468
C00891=1114.083,383.571,-89.212,-176.813,11.293,149.468
C00892=1114.079,383.819,-89.251,-176.811,11.295,149.467
C00893=1114.076,384.066,-89.288,-176.808,11.297,149.467
C00894=1114.072,384.313,-89.326,-176.805,11.300,149.467
C00895=1114.069,384.561,-89.363,-176.803,11.302,149.467
C00896=1114.065,384.807,-89.401,-176.800,11.305,149.467
C00897=1114.062,385.055,-89.439,-176.798,11.307,149.467
C00898=1114.057,385.301,-89.477,-176.795,11.310,149.468
C00899=1114.054,385.549,-89.515,-176.793,11.312,149.467
C00900=1114.050,385.796,-89.552,-176.790,11.315,149.467
C00901=1114.047,386.043,-89.590,-176.788,11.317,149.467
C00902=1114.042,386.290,-89.628,-176.786,11.320,149.468
C00903=1114.039,386.537,-89.666,-176.783,11.322,149.468
C00904=1114.035,386.784,-89.704,-176.780,11.325,149.468
C00905=1114.032,387.031,-89.742,-176.778,11.328,149.468
C00906=1114.028,387.278,-89.780,-176.776,11.330,149.468
C00907=1114.024,387.525,-89.818,-176.773,11.334,149.468
C00908=1114.021,387.773,-89.856,-176.770,11.336,149.468
C00909=1114.018,388.019,-89.893,-176.768,11.339,149.468
C00910=1114.014,388.267,-89.932,-176.766,11.342,149.468
C00911=1114.010,388.513,-89.969,-176.763,11.345,149.468
C00912=1114.007,388.725,-90.001,-176.761,11.347,149.468
C00913=1114.004,388.937,-90.035,-176.759,11.349,149.468
C00914=1114.001,389.148,-90.066,-176.757,11.352,149.469
C00915=1113.997,389.360,-90.099,-176.755,11.354,149.469
C00916=1113.995,389.571,-90.132,-176.753,11.356,149.469
C00917=1113.991,389.783,-90.164,-176.751,11.359,149.469
C00918=1113.988,389.994,-90.197,-176.749,11.362,149.469
C00919=1113.985,390.207,-90.230,-176.747,11.364,149.469
C00920=1113.982,390.454,-90.268,-176.744,11.367,149.469
C00921=1113.978,390.700,-90.307,-176.742,11.370,149.469
C00922=1113.974,390.948,-90.344,-176.739,11.373,149.470
C00923=1113.971,391.194,-90.382,-176.738,11.376,149.470
C00924=1113.967,391.442,-90.421,-176.735,11.379,149.470
C00925=1113.963,391.689,-90.459,-176.733,11.382,149.470
C00926=1113.959,391.936,-90.497,-176.730,11.386,149.471
C00927=1113.956,392.183,-90.535,-176.728,11.389,149.471
C00928=1113.953,392.430,-90.573,-176.726,11.392,149.471
C00929=1113.948,392.677,-90.611,-176.723,11.395,149.471
C00930=1113.945,392.924,-90.649,-176.721,11.398,149.471
C00931=1113.941,393.172,-90.688,-176.719,11.401,149.472
C00932=1113.938,393.418,-90.726,-176.717,11.404,149.472
C00933=1113.934,393.665,-90.765,-176.715,11.408,149.472
C00934=1113.931,393.912,-90.803,-176.712,11.411,149.472
C00935=1113.926,394.159,-90.842,-176.710,11.414,149.473
C00936=1113.923,394.406,-90.880,-176.708,11.418,149.473
C00937=1113.919,394.653,-90.918,-176.706,11.421,149.473
C00938=1113.916,394.900,-90.957,-176.703,11.425,149.474
C00939=1113.912,395.147,-90.995,-176.701,11.429,149.474
C00940=1113.909,395.394,-91.033,-176.699,11.432,149.475
C00941=1113.905,395.641,-91.072,-176.696,11.436,149.475
C00942=1113.901,395.888,-91.110,-176.694,11.439,149.475
C00943=1113.897,396.135,-91.148,-176.692,11.443,149.476
C00944=1113.895,396.382,-91.187,-176.690,11.446,149.476
C00945=1113.891,396.630,-91.225,-176.688,11.450,149.476
C00946=1113.887,396.876,-91.264,-176.686,11.453,149.477
C00947=1113.883,397.123,-91.302,-176.683,11.457,149.477
C00948=1113.880,397.370,-91.341,-176.681,11.461,149.478
C00949=1113.876,397.617,-91.379,-176.679,11.465,149.478
C00950=1113.872,397.864,-91.418,-176.677,11.468,149.479
C00951=1113.869,398.111,-91.456,-176.675,11.472,149.479
C00952=1113.865,398.358,-91.495,-176.673,11.476,149.479
C00953=1113.861,398.605,-91.534,-176.671,11.480,149.480
C00954=1113.859,398.852,-91.573,-176.669,11.483,149.480
C00955=1113.854,399.099,-91.611,-176.667,11.488,149.481
C00956=1113.851,399.346,-91.649,-176.665,11.491,149.481
C00957=1113.848,399.593,-91.689,-176.663,11.495,149.482
C00958=1113.844,399.840,-91.727,-176.660,11.500,149.483
C00959=1113.841,400.087,-91.766,-176.658,11.503,149.483
C00960=1113.836,400.334,-91.804,-176.656,11.508,149.484
C00961=1113.833,400.581,-91.843,-176.654,11.512,149.484
C00962=1113.830,400.827,-91.882,-176.652,11.516,149.485
C00963=1113.826,401.075,-91.921,-176.650,11.520,149.485
C00964=1113.822,401.322,-91.960,-176.648,11.524,149.486
C00965=1113.819,401.569,-91.999,-176.646,11.528,149.486
C00966=1113.815,401.815,-92.037,-176.644,11.532,149.487
C00967=1113.811,402.062,-92.076,-176.642,11.537,149.488
C00968=1113.808,402.274,-92.109,-176.641,11.541,149.488
C00969=1113.805,402.485,-92.143,-176.639,11.545,149.489
C00970=1113.803,402.697,-92.176,-176.637,11.549,149.489
C00971=1113.799,402.908,-92.209,-176.636,11.552,149.490
C00972=1113.796,403.120,-92.242,-176.634,11.556,149.491
C00973=1113.793,403.330,-92.276,-176.632,11.560,149.491
C00974=1113.790,403.542,-92.309,-176.630,11.564,149.492
C00975=1113.787,403.754,-92.343,-176.629,11.567,149.492
C00976=1113.784,404.000,-92.381,-176.627,11.572,149.493
C00977=1113.780,404.247,-92.421,-176.625,11.577,149.494
C00978=1113.776,404.494,-92.460,-176.623,11.581,149.494
C00979=1113.773,404.741,-92.499,-176.622,11.585,149.495
C00980=1113.769,404.989,-92.538,-176.620,11.590,149.496
C00981=1113.766,405.236,-92.576,-176.618,11.595,149.497
C00982=1113.762,405.483,-92.616,-176.616,11.600,149.497
C00983=1113.759,405.729,-92.655,-176.615,11.604,149.498
C00984=1113.755,405.976,-92.694,-176.613,11.609,149.499
C00985=1113.751,406.223,-92.733,-176.611,11.614,149.500
C00986=1113.747,406.470,-92.772,-176.609,11.619,149.501
C00987=1113.744,406.717,-92.811,-176.607,11.624,149.502
C00988=1113.741,406.963,-92.850,-176.605,11.629,149.502
C00989=1113.737,407.210,-92.889,-176.604,11.634,149.503
C00990=1113.734,407.457,-92.929,-176.602,11.639,149.504
C00991=1113.730,407.704,-92.968,-176.601,11.643,149.505
C00992=1113.726,407.951,-93.007,-176.599,11.648,149.506
C00993=1113.723,408.198,-93.046,-176.597,11.654,149.507
C00994=1113.719,408.444,-93.086,-176.595,11.659,149.508
C00995=1113.716,408.691,-93.126,-176.594,11.664,149.509
C00996=1113.712,408.938,-93.165,-176.591,11.670,149.510
C00997=1113.709,409.185,-93.204,-176.590,11.675,149.511
C00998=1113.705,409.432,-93.243,-176.588,11.680,149.511
C00999=1113.701,409.679,-93.283,-176.587,11.685,149.512
C01000=1113.698,409.926,-93.323,-176.585,11.691,149.513
C01001=1113.694,410.173,-93.362,-176.584,11.696,149.515
C01002=1113.691,410.419,-93.401,-176.582,11.701,149.516
C01003=1113.688,410.667,-93.441,-176.581,11.707,149.517
C01004=1113.684,410.914,-93.480,-176.578,11.713,149.518
C01005=1113.681,411.160,-93.520,-176.577,11.718,149.519
C01006=1113.677,411.407,-93.559,-176.576,11.723,149.520
C01007=1113.674,411.654,-93.598,-176.574,11.729,149.521
C01008=1113.670,411.901,-93.638,-176.572,11.735,149.522
C01009=1113.667,412.148,-93.678,-176.571,11.740,149.523
C01010=1113.663,412.395,-93.717,-176.570,11.746,149.524
C01011=1113.660,412.641,-93.757,-176.568,11.752,149.525
C01012=1113.656,412.888,-93.796,-176.567,11.758,149.527
C01013=1113.652,413.135,-93.835,-176.566,11.763,149.528
C01014=1113.649,413.381,-93.875,-176.564,11.770,149.529
C01015=1113.646,413.629,-93.915,-176.563,11.775,149.530
C01016=1113.643,413.875,-93.955,-176.561,11.782,149.531
C01017=1113.641,414.122,-93.995,-176.560,11.787,149.532
C01018=1113.639,414.369,-94.033,-176.558,11.794,149.534
C01019=1113.638,414.616,-94.073,-176.557,11.799,149.535
C01020=1113.637,414.863,-94.112,-176.555,11.806,149.536
C01021=1113.637,415.110,-94.151,-176.554,11.812,149.537
C01022=1113.638,415.357,-94.191,-176.553,11.818,149.539
C01023=1113.638,415.603,-94.230,-176.552,11.824,149.540
C01024=1113.639,415.814,-94.264,-176.550,11.829,149.541
C01025=1113.641,416.026,-94.297,-176.549,11.835,149.542
C01026=1113.643,416.237,-94.331,-176.549,11.840,149.543
C01027=1113.645,416.448,-94.364,-176.547,11.845,149.545
C01028=1113.648,416.659,-94.397,-176.546,11.851,149.546
C01029=1113.650,416.871,-94.430,-176.545,11.857,149.547
C01030=1113.653,417.082,-94.463,-176.545,11.861,149.548
C01031=1113.658,417.293,-94.496,-176.544,11.867,149.550
C01032=1113.239,417.292,-94.559,-176.536,11.872,149.549
C01033=1113.235,417.081,-94.525,-176.537,11.866,149.548
C01034=1113.232,416.871,-94.493,-176.538,11.861,149.546
C01035=1113.229,416.659,-94.459,-176.539,11.855,149.545
C01036=1113.226,416.448,-94.426,-176.540,11.850,149.544
C01037=1113.224,416.236,-94.393,-176.541,11.844,149.543
C01038=1113.222,416.026,-94.360,-176.542,11.839,149.542
C01039=1113.221,415.814,-94.326,-176.543,11.834,149.540
C01040=1113.219,415.603,-94.293,-176.545,11.828,149.539
C01041=1113.218,415.356,-94.254,-176.546,11.822,149.538
C01042=1113.218,415.110,-94.214,-176.547,11.816,149.537
C01043=1113.218,414.863,-94.175,-176.549,11.810,149.536
C01044=1113.218,414.616,-94.135,-176.550,11.804,149.534
C01045=1113.220,414.369,-94.096,-176.551,11.797,149.533
C01046=1113.222,414.123,-94.057,-176.553,11.792,149.532
C01047=1113.224,413.875,-94.018,-176.554,11.786,149.531
C01048=1113.227,413.628,-93.977,-176.555,11.780,149.529
C01049=1113.230,413.382,-93.937,-176.557,11.773,149.528
C01050=1113.233,413.135,-93.898,-176.558,11.768,149.527
C01051=1113.237,412.888,-93.859,-176.560,11.761,149.526
C01052=1113.240,412.642,-93.819,-176.562,11.756,149.525
C01053=1113.243,412.394,-93.779,-176.563,11.750,149.524
C01054=1113.247,412.148,-93.739,-176.565,11.744,149.522
C01055=1113.250,411.901,-93.700,-176.567,11.738,149.521
C01056=1113.255,411.653,-93.660,-176.568,11.733,149.520
C01057=1113.258,411.407,-93.620,-176.569,11.727,149.519
C01058=1113.262,411.160,-93.581,-176.572,11.721,149.518
C01059=1113.265,410.913,-93.542,-176.573,11.716,149.517
C01060=1113.269,410.666,-93.502,-176.574,11.710,149.516
C01061=1113.272,410.420,-93.462,-176.576,11.705,149.515
C01062=1113.276,410.173,-93.423,-176.578,11.699,149.514
C01063=1113.279,409.926,-93.384,-176.580,11.694,149.513
C01064=1113.283,409.679,-93.345,-176.581,11.689,149.512
C01065=1113.286,409.433,-93.305,-176.583,11.684,149.511
C01066=1113.290,409.186,-93.266,-176.584,11.678,149.510
C01067=1113.294,408.939,-93.226,-176.586,11.673,149.509
C01068=1113.297,408.692,-93.187,-176.588,11.667,149.508
C01069=1113.301,408.445,-93.148,-176.590,11.662,149.507
C01070=1113.304,408.198,-93.109,-176.592,11.657,149.506
C01071=1113.307,407.952,-93.069,-176.593,11.652,149.505
C01072=1113.311,407.705,-93.030,-176.595,11.647,149.505
C01073=1113.314,407.458,-92.991,-176.597,11.642,149.504
C01074=1113.318,407.211,-92.951,-176.599,11.637,149.503
C01075=1113.322,406.964,-92.912,-176.600,11.632,149.502
C01076=1113.325,406.717,-92.873,-176.602,11.627,149.501
C01077=1113.329,406.470,-92.834,-176.604,11.622,149.500
C01078=1113.332,406.223,-92.794,-176.606,11.616,149.499
C01079=1113.335,405.976,-92.756,-176.607,11.612,149.499
C01080=1113.339,405.729,-92.716,-176.609,11.607,149.498
C01081=1113.342,405.482,-92.677,-176.611,11.603,149.497
C01082=1113.346,405.235,-92.638,-176.613,11.598,149.496
C01083=1113.350,404.989,-92.599,-176.615,11.593,149.495
C01084=1113.353,404.742,-92.559,-176.617,11.588,149.495
C01085=1113.356,404.495,-92.521,-176.619,11.584,149.494
C01086=1113.360,404.248,-92.482,-176.621,11.579,149.493
C01087=1113.364,404.000,-92.443,-176.623,11.574,149.492
C01088=1113.367,403.753,-92.404,-176.625,11.570,149.492
C01089=1113.371,403.543,-92.370,-176.627,11.566,149.491
C01090=1113.374,403.331,-92.337,-176.628,11.562,149.491
C01091=1113.376,403.120,-92.304,-176.630,11.558,149.490
C01092=1113.380,402.908,-92.271,-176.632,11.554,149.489
C01093=1113.382,402.697,-92.237,-176.633,11.550,149.489
C01094=1113.386,402.485,-92.204,-176.635,11.547,149.488
C01095=1113.389,402.274,-92.170,-176.637,11.543,149.488
C01096=1113.392,402.062,-92.137,-176.638,11.539,149.487
C01097=1113.395,401.816,-92.099,-176.640,11.535,149.487
C01098=1113.399,401.569,-92.059,-176.642,11.531,149.486
C01099=1113.403,401.321,-92.021,-176.644,11.527,149.485
C01100=1113.406,401.075,-91.982,-176.647,11.522,149.485
C01101=1113.410,400.828,-91.943,-176.648,11.518,149.484
C01102=1113.413,400.581,-91.904,-176.651,11.514,149.484
C01103=1113.418,400.334,-91.865,-176.652,11.510,149.483
C01104=1113.421,400.087,-91.827,-176.655,11.505,149.483
C01105=1113.424,399.840,-91.788,-176.657,11.502,149.482
C01106=1113.428,399.593,-91.749,-176.659,11.497,149.482
C01107=1113.431,399.346,-91.710,-176.661,11.494,149.481
C01108=1113.435,399.099,-91.672,-176.663,11.490,149.481
C01109=1113.438,398.853,-91.634,-176.665,11.486,149.480
C01110=1113.442,398.605,-91.595,-176.667,11.482,149.480
C01111=1113.446,398.358,-91.556,-176.669,11.478,149.479
C01112=1113.449,398.111,-91.517,-176.672,11.474,149.479
C01113=1113.453,397.865,-91.479,-176.674,11.470,149.478
C01114=1113.457,397.618,-91.440,-176.676,11.467,149.478
C01115=1113.460,397.370,-91.402,-176.678,11.463,149.477
C01116=1113.464,397.123,-91.363,-176.681,11.459,149.477
C01117=1113.467,396.876,-91.325,-176.683,11.456,149.477
C01118=1113.471,396.630,-91.286,-176.684,11.452,149.476
C01119=1113.474,396.383,-91.248,-176.687,11.448,149.476
C01120=1113.478,396.135,-91.209,-176.689,11.444,149.475
C01121=1113.482,395.888,-91.170,-176.691,11.441,149.475
C01122=1113.486,395.641,-91.132,-176.694,11.437,149.475
C01123=1113.489,395.394,-91.093,-176.696,11.434,149.474
C01124=1113.492,395.147,-91.055,-176.698,11.430,149.474
C01125=1113.497,394.900,-91.017,-176.700,11.427,149.474
C01126=1113.500,394.654,-90.978,-176.703,11.423,149.473
C01127=1113.504,394.406,-90.940,-176.705,11.420,149.473
C01128=1113.507,394.159,-90.902,-176.707,11.416,149.473
C01129=1113.511,393.913,-90.863,-176.710,11.413,149.472
C01130=1113.514,393.665,-90.825,-176.712,11.410,149.472
C01131=1113.518,393.418,-90.787,-176.714,11.406,149.472
C01132=1113.522,393.172,-90.748,-176.717,11.403,149.472
C01133=1113.526,392.924,-90.710,-176.719,11.399,149.471
C01134=1113.529,392.677,-90.672,-176.721,11.396,149.471
C01135=1113.533,392.430,-90.634,-176.724,11.393,149.471
C01136=1113.536,392.183,-90.595,-176.726,11.390,149.470
C01137=1113.540,391.936,-90.557,-176.728,11.386,149.470
C01138=1113.544,391.689,-90.519,-176.731,11.383,149.470
C01139=1113.547,391.442,-90.481,-176.733,11.381,149.470
C01140=1113.550,391.195,-90.443,-176.735,11.378,149.470
C01141=1113.555,390.948,-90.405,-176.738,11.375,149.470
C01142=1113.558,390.701,-90.366,-176.740,11.372,149.469
C01143=1113.562,390.454,-90.328,-176.743,11.368,149.469
C01144=1113.566,390.207,-90.290,-176.745,11.365,149.469
C01145=1113.568,389.995,-90.258,-176.747,11.363,149.469
C01146=1113.572,389.784,-90.225,-176.749,11.361,149.469
C01147=1113.574,389.573,-90.192,-176.751,11.358,149.469
C01148=1113.578,389.360,-90.160,-176.753,11.355,149.468
C01149=1113.580,389.149,-90.127,-176.755,11.353,149.468
C01150=1113.584,388.937,-90.095,-176.757,11.350,149.468
C01151=1113.587,388.726,-90.062,-176.759,11.348,149.468
C01152=1113.591,388.515,-90.029,-176.762,11.345,149.468
C01153=1113.594,388.268,-89.991,-176.764,11.343,149.468
C01154=1113.597,388.020,-89.953,-176.767,11.340,149.468
C01155=1113.602,387.773,-89.915,-176.769,11.337,149.468
C01156=1113.605,387.525,-89.878,-176.771,11.335,149.468
C01157=1113.609,387.279,-89.840,-176.774,11.332,149.468
C01158=1113.612,387.032,-89.802,-176.777,11.329,149.468
C01159=1113.616,386.784,-89.764,-176.779,11.326,149.467
C01160=1113.620,386.538,-89.726,-176.782,11.324,149.467
C01161=1113.623,386.290,-89.688,-176.784,11.321,149.467
C01162=1113.627,386.044,-89.651,-176.786,11.318,149.467
C01163=1113.631,385.796,-89.612,-176.789,11.316,149.467
C01164=1113.634,385.550,-89.575,-176.792,11.314,149.467
C01165=1113.638,385.302,-89.537,-176.794,11.310,149.467
C01166=1113.641,385.056,-89.499,-176.796,11.308,149.467
C01167=1113.646,384.807,-89.461,-176.799,11.306,149.467
C01168=1113.649,384.561,-89.424,-176.801,11.304,149.467
C01169=1113.653,384.314,-89.386,-176.804,11.301,149.467
C01170=1113.656,384.067,-89.348,-176.807,11.299,149.467
C01171=1113.660,383.820,-89.310,-176.810,11.296,149.467
C01172=1113.664,383.573,-89.274,-176.812,11.294,149.467
C01173=1113.668,383.325,-89.235,-176.815,11.291,149.467
C01174=1113.671,383.078,-89.197,-176.818,11.289,149.468
C01175=1113.675,382.831,-89.159,-176.821,11.286,149.468
C01176=1113.679,382.584,-89.123,-176.824,11.283,149.468
C01177=1113.682,382.337,-89.085,-176.827,11.280,149.468
C01178=1113.686,382.090,-89.047,-176.830,11.278,149.468
C01179=1113.689,381.842,-89.010,-176.834,11.275,149.468
C01180=1113.694,381.595,-88.972,-176.837,11.272,149.468
C01181=1113.697,381.348,-88.934,-176.840,11.269,149.468
C01182=1113.701,381.101,-88.897,-176.844,11.267,149.469
C01183=1113.704,380.854,-88.859,-176.847,11.264,149.469
C01184=1113.708,380.607,-88.821,-176.850,11.262,149.469
C01185=1113.712,380.360,-88.785,-176.853,11.259,149.469
C01186=1113.715,380.113,-88.747,-176.856,11.256,149.469
C01187=1113.719,379.865,-88.710,-176.859,11.254,149.469
C01188=1113.723,379.618,-88.672,-176.863,11.251,149.469
C01189=1113.727,379.371,-88.635,-176.866,11.249,149.470
C01190=1113.730,379.124,-88.597,-176.869,11.246,149.470
C01191=1113.734,378.876,-88.560,-176.872,11.244,149.470
C01192=1113.738,378.630,-88.523,-176.875,11.241,149.470
C01193=1113.741,378.382,-88.485,-176.879,11.239,149.470
C01194=1113.745,378.135,-88.448,-176.882,11.236,149.470
C01195=1113.749,377.888,-88.411,-176.885,11.233,149.470
C01196=1113.752,377.641,-88.373,-176.888,11.231,149.471
C01197=1113.756,377.394,-88.336,-176.892,11.228,149.471
C01198=1113.760,377.146,-88.299,-176.895,11.226,149.471
C01199=1113.764,376.899,-88.261,-176.898,11.223,149.471
C01200=1113.768,376.652,-88.224,-176.901,11.221,149.471
C01201=1113.770,376.440,-88.192,-176.904,11.218,149.471
C01202=1113.774,376.229,-88.161,-176.907,11.216,149.472
C01203=1113.777,376.017,-88.129,-176.910,11.214,149.472
C01204=1113.780,375.805,-88.097,-176.913,11.212,149.472
C01205=1113.784,375.594,-88.065,-176.915,11.210,149.472
C01206=1113.787,375.382,-88.033,-176.919,11.208,149.472
C01207=1113.790,375.170,-88.002,-176.921,11.206,149.472
C01208=1113.793,374.958,-87.970,-176.924,11.203,149.473
C01209=1113.797,374.711,-87.933,-176.927,11.201,149.473
C01210=1113.801,374.464,-87.896,-176.931,11.198,149.473
C01211=1113.804,374.217,-87.859,-176.934,11.196,149.473
C01212=1113.808,373.969,-87.822,-176.937,11.193,149.473
C01213=1113.812,373.722,-87.785,-176.941,11.191,149.474
C01214=1113.815,373.475,-87.747,-176.944,11.188,149.474
C01215=1113.819,373.228,-87.711,-176.947,11.186,149.474
C01216=1113.823,372.980,-87.674,-176.950,11.183,149.474
C01217=1113.827,372.734,-87.637,-176.954,11.181,149.474
C01218=1113.830,372.486,-87.600,-176.957,11.178,149.475
C01219=1113.834,372.239,-87.563,-176.960,11.176,149.475
C01220=1113.838,371.991,-87.526,-176.964,11.173,149.475
C01221=1113.842,371.744,-87.490,-176.967,11.171,149.475
C01222=1113.845,371.497,-87.453,-176.970,11.168,149.475
C01223=1113.849,371.249,-87.416,-176.974,11.166,149.476
C01224=1113.853,371.002,-87.379,-176.977,11.163,149.476
C01225=1113.857,370.755,-87.343,-176.980,11.162,149.476
C01226=1113.861,370.508,-87.306,-176.983,11.160,149.477
C01227=1113.864,370.260,-87.269,-176.987,11.157,149.477
C01228=1113.868,370.013,-87.233,-176.990,11.155,149.477
C01229=1113.872,369.766,-87.196,-176.993,11.152,149.477
C01230=1113.876,369.519,-87.159,-176.996,11.150,149.477
C01231=1113.879,369.272,-87.123,-177.000,11.147,149.478
C01232=1113.883,369.024,-87.085,-177.003,11.145,149.478
C01233=1113.887,368.777,-87.049,-177.006,11.142,149.478
C01234=1113.890,368.530,-87.012,-177.010,11.140,149.478
C01235=1113.894,368.283,-86.975,-177.013,11.138,149.479
C01236=1113.898,368.036,-86.939,-177.017,11.135,149.479
C01237=1113.902,367.788,-86.903,-177.020,11.133,149.479
C01238=1113.905,367.540,-86.866,-177.023,11.130,149.479
C01239=1113.909,367.293,-86.830,-177.027,11.128,149.479
C01240=1113.913,367.046,-86.793,-177.030,11.126,149.480
C01241=1113.917,366.799,-86.756,-177.034,11.123,149.480
C01242=1113.921,366.552,-86.720,-177.037,11.121,149.480
C01243=1113.925,366.304,-86.683,-177.040,11.118,149.480
C01244=1113.928,366.058,-86.647,-177.043,11.116,149.481
C01245=1113.933,365.810,-86.611,-177.047,11.114,149.481
C01246=1113.935,365.562,-86.574,-177.050,11.111,149.481
C01247=1113.939,365.315,-86.538,-177.054,11.109,149.481
C01248=1113.943,365.068,-86.501,-177.057,11.106,149.482
C01249=1113.947,364.820,-86.465,-177.060,11.104,149.482
C01250=1113.950,364.573,-86.429,-177.064,11.102,149.482
C01251=1113.955,364.326,-86.393,-177.067,11.099,149.482
C01252=1113.958,364.079,-86.357,-177.071,11.097,149.483
C01253=1113.962,363.831,-86.320,-177.074,11.094,149.483
C01254=1113.966,363.584,-86.284,-177.077,11.092,149.483
C01255=1113.970,363.337,-86.247,-177.081,11.089,149.484
C01256=1113.974,363.089,-86.212,-177.084,11.087,149.484
C01257=1113.976,362.877,-86.180,-177.087,11.085,149.484
C01258=1113.980,362.665,-86.149,-177.090,11.084,149.484
C01259=1113.983,362.454,-86.118,-177.093,11.081,149.484
C01260=1113.987,362.242,-86.088,-177.095,11.079,149.485
C01261=1113.990,362.029,-86.056,-177.098,11.077,149.485
C01262=1113.992,361.818,-86.025,-177.101,11.075,149.485
C01263=1113.996,361.606,-85.994,-177.104,11.073,149.485
C01264=1114.000,361.394,-85.963,-177.107,11.071,149.485
C01265=1114.003,361.147,-85.928,-177.110,11.068,149.486
C01266=1114.007,360.900,-85.891,-177.114,11.066,149.486
C01267=1114.011,360.652,-85.855,-177.117,11.064,149.486
C01268=1114.014,360.405,-85.819,-177.121,11.061,149.487
C01269=1114.019,360.157,-85.783,-177.124,11.059,149.487
C01270=1114.022,359.910,-85.748,-177.127,11.056,149.487
C01271=1114.026,359.663,-85.711,-177.131,11.054,149.487
C01272=1114.029,359.415,-85.676,-177.134,11.052,149.488
C01273=1114.034,359.168,-85.640,-177.138,11.049,149.488
C01274=1114.037,358.921,-85.603,-177.141,11.047,149.488
C01275=1114.041,358.673,-85.568,-177.144,11.044,149.488
C01276=1114.045,358.425,-85.532,-177.148,11.042,149.488
C01277=1114.049,358.178,-85.496,-177.151,11.040,149.489
C01278=1114.052,357.931,-85.460,-177.155,11.037,149.489
C01279=1114.056,357.684,-85.424,-177.158,11.035,149.489
C01280=1114.060,357.436,-85.388,-177.161,11.032,149.489
C01281=1114.064,357.188,-85.353,-177.165,11.030,149.490
C01282=1114.068,356.941,-85.317,-177.168,11.028,149.490
C01283=1114.071,356.694,-85.281,-177.172,11.025,149.490
C01284=1114.075,356.447,-85.246,-177.175,11.023,149.491
C01285=1114.080,356.199,-85.209,-177.178,11.020,149.491
C01286=1114.083,355.952,-85.174,-177.181,11.018,149.491
C01287=1114.087,355.704,-85.138,-177.185,11.015,149.491
C01288=1114.091,355.457,-85.103,-177.188,11.013,149.492
C01289=1114.094,355.209,-85.067,-177.192,11.011,149.492
C01290=1114.098,354.962,-85.032,-177.195,11.008,149.492
C01291=1114.102,354.714,-84.996,-177.198,11.006,149.492
C01292=1114.107,354.467,-84.960,-177.202,11.003,149.493
C01293=1114.110,354.220,-84.925,-177.205,11.001,149.493
C01294=1114.114,353.972,-84.889,-177.208,10.998,149.493
C01295=1114.118,353.725,-84.854,-177.212,10.996,149.493
C01296=1114.121,353.477,-84.818,-177.215,10.994,149.494
C01297=1114.125,353.230,-84.783,-177.219,10.991,149.494
C01298=1114.129,352.983,-84.747,-177.222,10.989,149.494
C01299=1114.133,352.735,-84.712,-177.225,10.986,149.494
C01300=1114.137,352.488,-84.676,-177.229,10.984,149.494
C01301=1114.140,352.240,-84.641,-177.232,10.982,149.495
C01302=1114.144,351.993,-84.605,-177.235,10.979,149.495
C01303=1114.148,351.745,-84.570,-177.239,10.977,149.495
C01304=1114.153,351.498,-84.534,-177.242,10.974,149.495
C01305=1114.157,351.250,-84.499,-177.245,10.972,149.496
C01306=1114.160,351.003,-84.464,-177.249,10.968,149.496
C01307=1114.164,350.755,-84.428,-177.252,10.966,149.496
C01308=1114.168,350.508,-84.393,-177.256,10.964,149.496
C01309=1114.172,350.261,-84.357,-177.259,10.961,149.496
C01310=1114.175,350.013,-84.323,-177.262,10.959,149.497
C01311=1114.179,349.766,-84.287,-177.266,10.956,149.497
C01312=1114.183,349.519,-84.252,-177.269,10.954,149.497
C01313=1114.187,349.306,-84.222,-177.272,10.952,149.497
C01314=1114.190,349.095,-84.192,-177.275,10.950,149.498
C01315=1114.193,348.882,-84.162,-177.277,10.948,149.498
C01316=1114.197,348.670,-84.131,-177.280,10.946,149.498
C01317=1114.200,348.458,-84.102,-177.283,10.943,149.498
C01318=1114.203,348.246,-84.071,-177.285,10.941,149.498
C01319=1114.207,348.034,-84.041,-177.289,10.939,149.498
C01320=1114.210,347.822,-84.011,-177.291,10.937,149.499
C01321=1114.214,347.574,-83.976,-177.294,10.934,149.499
C01322=1114.217,347.327,-83.940,-177.298,10.932,149.499
C01323=1114.222,347.079,-83.906,-177.301,10.930,149.499
C01324=1114.226,346.832,-83.870,-177.304,10.927,149.499
C01325=1114.229,346.584,-83.836,-177.307,10.925,149.500
C01326=1114.233,346.337,-83.801,-177.310,10.923,149.500
C01327=1114.237,346.090,-83.766,-177.313,10.920,149.500
C01328=1114.241,345.841,-83.731,-177.317,10.918,149.500
C01329=1114.245,345.595,-83.696,-177.320,10.915,149.500
C01330=1114.249,345.347,-83.661,-177.323,10.912,149.501
C01331=1114.252,345.099,-83.626,-177.326,10.910,149.501
C01332=1114.256,344.852,-83.591,-177.329,10.908,149.501
C01333=1114.260,344.604,-83.556,-177.333,10.905,149.501
C01334=1114.265,344.357,-83.521,-177.336,10.903,149.501
C01335=1114.269,344.109,-83.486,-177.339,10.900,149.501
C01336=1114.272,343.862,-83.451,-177.342,10.898,149.502
C01337=1114.276,343.614,-83.417,-177.345,10.896,149.502
C01338=1114.280,343.366,-83.382,-177.348,10.893,149.502
C01339=1114.284,343.119,-83.347,-177.352,10.891,149.502
C01340=1114.288,342.872,-83.313,-177.354,10.888,149.502
C01341=1114.292,342.623,-83.278,-177.358,10.885,149.503
C01342=1114.296,342.377,-83.243,-177.361,10.883,149.503
C01343=1114.299,342.129,-83.208,-177.364,10.881,149.503
C01344=1114.304,341.881,-83.174,-177.368,10.878,149.503
C01345=1114.307,341.634,-83.138,-177.371,10.875,149.503
C01346=1114.312,341.387,-83.104,-177.374,10.873,149.504
C01347=1114.315,341.139,-83.070,-177.377,10.871,149.504
C01348=1114.319,340.891,-83.035,-177.380,10.869,149.504
C01349=1114.324,340.643,-83.000,-177.383,10.866,149.504
C01350=1114.327,340.396,-82.966,-177.386,10.864,149.504
C01351=1114.331,340.149,-82.931,-177.390,10.861,149.505
C01352=1114.335,339.900,-82.896,-177.393,10.859,149.505
C01353=1114.339,339.653,-82.862,-177.396,10.856,149.505
C01354=1114.343,339.405,-82.828,-177.399,10.853,149.505
C01355=1114.347,339.158,-82.794,-177.402,10.851,149.505
C01356=1114.351,338.910,-82.759,-177.406,10.848,149.506
C01357=1114.355,338.663,-82.724,-177.409,10.846,149.506
C01358=1114.358,338.415,-82.689,-177.412,10.844,149.506
C01359=1114.363,338.168,-82.655,-177.415,10.842,149.506
C01360=1114.366,337.920,-82.621,-177.418,10.839,149.506
C01361=1114.371,337.673,-82.586,-177.421,10.837,149.507
C01362=1114.374,337.425,-82.552,-177.425,10.834,149.507
C01363=1114.378,337.177,-82.518,-177.427,10.831,149.507
C01364=1114.382,336.930,-82.484,-177.431,10.829,149.507
C01365=1114.386,336.682,-82.449,-177.434,10.826,149.507
C01366=1114.390,336.435,-82.415,-177.437,10.824,149.508
C01367=1114.394,336.187,-82.380,-177.440,10.821,149.508
C01368=1114.398,335.940,-82.346,-177.444,10.819,149.508
C01369=1114.401,335.728,-82.317,-177.446,10.817,149.508
C01370=1114.404,335.515,-82.288,-177.449,10.815,149.508
C01371=1114.408,335.303,-82.258,-177.452,10.812,149.508
C01372=1114.412,335.091,-82.229,-177.454,10.811,149.509
C01373=1114.415,334.879,-82.199,-177.457,10.809,149.509
C01374=1114.418,334.666,-82.170,-177.460,10.806,149.509
C01375=1114.421,334.454,-82.141,-177.462,10.804,149.509
C01376=1114.425,334.242,-82.112,-177.465,10.803,149.509
C01377=1114.429,333.994,-82.077,-177.468,10.800,149.510
C01378=1114.432,333.747,-82.043,-177.471,10.797,149.510
C01379=1114.437,333.498,-82.009,-177.474,10.795,149.510
C01380=1114.440,333.251,-81.976,-177.478,10.792,149.510
C01381=1114.445,333.004,-81.941,-177.481,10.790,149.510
C01382=1114.448,332.756,-81.907,-177.484,10.787,149.510
C01383=1114.452,332.509,-81.873,-177.487,10.785,149.511
C01384=1114.457,332.261,-81.839,-177.491,10.782,149.511
C01385=1114.460,332.013,-81.805,-177.494,10.779,149.511
C01386=1114.464,331.766,-81.771,-177.497,10.777,149.511
C01387=1114.468,331.517,-81.737,-177.500,10.775,149.511
C01388=1114.472,331.270,-81.703,-177.502,10.773,149.512
C01389=1114.476,331.023,-81.669,-177.506,10.770,149.512
C01390=1114.480,330.774,-81.635,-177.509,10.768,149.512
C01391=1114.484,330.527,-81.601,-177.512,10.765,149.512
C01392=1114.488,330.280,-81.567,-177.515,10.762,149.512
C01393=1114.491,330.032,-81.534,-177.519,10.760,149.513
C01394=1114.496,329.784,-81.499,-177.522,10.758,149.513
C01395=1114.500,329.536,-81.466,-177.525,10.755,149.513
C01396=1114.504,329.289,-81.432,-177.528,10.752,149.513
C01397=1114.508,329.041,-81.399,-177.532,10.750,149.513
C01398=1114.512,328.794,-81.364,-177.534,10.748,149.513
C01399=1114.516,328.546,-81.331,-177.537,10.745,149.514
C01400=1114.519,328.298,-81.297,-177.540,10.743,149.514
C01401=1114.524,328.050,-81.264,-177.543,10.740,149.514
C01402=1114.527,327.803,-81.230,-177.547,10.738,149.514
C01403=1114.532,327.555,-81.196,-177.550,10.735,149.514
C01404=1114.536,327.307,-81.162,-177.553,10.733,149.515
C01405=1114.540,327.060,-81.129,-177.556,10.730,149.515
C01406=1114.543,326.812,-81.095,-177.560,10.728,149.515
C01407=1114.548,326.565,-81.062,-177.563,10.725,149.515
C01408=1114.551,326.316,-81.028,-177.566,10.722,149.515
C01409=1114.556,326.069,-80.994,-177.569,10.720,149.516
C01410=1114.560,325.821,-80.961,-177.572,10.718,149.516
C01411=1114.564,325.574,-80.927,-177.575,10.715,149.516
C01412=1114.567,325.326,-80.893,-177.578,10.713,149.516
C01413=1114.571,325.078,-80.860,-177.581,10.711,149.516
C01414=1114.576,324.830,-80.827,-177.584,10.708,149.516
C01415=1114.579,324.583,-80.793,-177.588,10.705,149.517
C01416=1114.583,324.335,-80.760,-177.591,10.703,149.517
C01417=1114.587,324.087,-80.726,-177.594,10.700,149.517
C01418=1114.591,323.840,-80.692,-177.597,10.698,149.517
C01419=1114.595,323.592,-80.659,-177.600,10.695,149.517
C01420=1114.599,323.344,-80.626,-177.603,10.692,149.518
C01421=1114.603,323.097,-80.593,-177.606,10.691,149.518
C01422=1114.607,322.848,-80.559,-177.609,10.688,149.518
C01423=1114.611,322.601,-80.526,-177.612,10.686,149.518
C01424=1114.615,322.353,-80.492,-177.616,10.683,149.518
C01425=1114.619,322.141,-80.464,-177.619,10.680,149.518
C01426=1114.622,321.929,-80.436,-177.621,10.678,149.519
C01427=1114.625,321.716,-80.407,-177.624,10.677,149.519
C01428=1114.629,321.504,-80.379,-177.627,10.674,149.519
C01429=1114.632,321.291,-80.350,-177.629,10.672,149.519
C01430=1114.635,321.079,-80.322,-177.632,10.670,149.519
C01431=1114.639,320.867,-80.292,-177.634,10.667,149.519
C01432=1114.642,320.655,-80.265,-177.637,10.666,149.520
C01433=1114.646,320.407,-80.231,-177.640,10.663,149.520
C01434=1114.650,320.160,-80.198,-177.643,10.661,149.520
C01435=1114.654,319.911,-80.165,-177.647,10.658,149.520
C01436=1114.658,319.663,-80.132,-177.650,10.655,149.520
C01437=1114.662,319.416,-80.098,-177.653,10.653,149.520
C01438=1114.666,319.168,-80.065,-177.656,10.651,149.521
C01439=1114.670,318.920,-80.032,-177.659,10.648,149.521
C01440=1114.674,318.673,-80.000,-177.662,10.646,149.521
C01441=1114.678,318.425,-79.966,-177.665,10.643,149.521
C01442=1114.682,318.177,-79.933,-177.668,10.641,149.521
C01443=1114.687,317.929,-79.901,-177.672,10.638,149.522
C01444=1114.691,317.681,-79.868,-177.674,10.636,149.522
C01445=1114.695,317.434,-79.834,-177.678,10.633,149.522
C01446=1114.698,317.186,-79.802,-177.681,10.630,149.522
C01447=1114.702,316.938,-79.769,-177.684,10.628,149.522
C01448=1114.707,316.691,-79.736,-177.687,10.626,149.523
C01449=1114.710,316.442,-79.702,-177.690,10.623,149.523
C01450=1114.714,316.194,-79.670,-177.693,10.621,149.523
C01451=1114.718,315.946,-79.637,-177.696,10.618,149.523
C01452=1114.722,315.699,-79.604,-177.699,10.616,149.523
C01453=1114.726,315.451,-79.571,-177.703,10.613,149.523
C01454=1114.730,315.203,-79.539,-177.705,10.611,149.524
C01455=1114.734,314.955,-79.506,-177.709,10.608,149.524
C01456=1114.738,314.707,-79.473,-177.712,10.605,149.524
C01457=1114.742,314.460,-79.439,-177.715,10.603,149.524
C01458=1114.746,314.212,-79.408,-177.718,10.601,149.524
C01459=1114.750,313.964,-79.374,-177.721,10.599,149.524
C01460=1114.754,313.716,-79.341,-177.724,10.596,149.525
C01461=1114.759,313.469,-79.310,-177.727,10.593,149.525
C01462=1114.763,313.221,-79.277,-177.730,10.591,149.525
C01463=1114.767,312.973,-79.243,-177.733,10.588,149.525
C01464=1114.771,312.725,-79.212,-177.737,10.586,149.525
C01465=1114.775,312.478,-79.178,-177.740,10.583,149.526
C01466=1114.779,312.229,-79.146,-177.743,10.580,149.526
C01467=1114.783,311.982,-79.113,-177.746,10.578,149.526
C01468=1114.787,311.734,-79.080,-177.749,10.575,149.526
C01469=1114.790,311.486,-79.048,-177.752,10.573,149.526
C01470=1114.795,311.238,-79.015,-177.755,10.571,149.526
C01471=1114.799,310.990,-78.983,-177.758,10.568,149.527
C01472=1114.802,310.743,-78.950,-177.761,10.566,149.527
C01473=1114.807,310.494,-78.918,-177.764,10.563,149.527
C01474=1114.810,310.247,-78.885,-177.768,10.561,149.527
C01475=1114.815,309.999,-78.853,-177.770,10.558,149.527
C01476=1114.819,309.752,-78.820,-177.774,10.556,149.528
C01477=1114.823,309.503,-78.788,-177.777,10.553,149.528
C01478=1114.828,309.255,-78.756,-177.780,10.550,149.528
C01479=1114.831,309.008,-78.723,-177.783,10.548,149.528
C01480=1114.835,308.759,-78.691,-177.786,10.546,149.528
C01481=1114.839,308.547,-78.663,-177.789,10.543,149.528
C01482=1114.842,308.335,-78.636,-177.791,10.541,149.529
C01483=1114.846,308.122,-78.608,-177.794,10.539,149.529
C01484=1114.849,307.910,-78.580,-177.797,10.537,149.529
C01485=1114.853,307.697,-78.553,-177.799,10.535,149.529
C01486=1114.856,307.485,-78.524,-177.802,10.532,149.529
C01487=1114.860,307.272,-78.497,-177.804,10.530,149.529
C01488=1114.864,307.060,-78.470,-177.807,10.529,149.530
C01489=1114.867,306.812,-78.437,-177.810,10.526,149.530
C01490=1114.871,306.564,-78.405,-177.813,10.523,149.530
C01491=1114.875,306.316,-78.373,-177.816,10.521,149.530
C01492=1114.880,306.068,-78.341,-177.820,10.518,149.530
C01493=1114.884,305.821,-78.308,-177.823,10.515,149.530
C01494=1114.887,305.573,-78.276,-177.826,10.513,149.531
C01495=1114.892,305.324,-78.244,-177.829,10.510,149.531
C01496=1114.896,305.077,-78.212,-177.832,10.509,149.531
C01497=1114.900,304.829,-78.180,-177.835,10.506,149.531
C01498=1114.904,304.581,-78.147,-177.838,10.503,149.531
C01499=1114.908,304.333,-78.116,-177.841,10.501,149.531
C01500=1114.912,304.085,-78.083,-177.844,10.498,149.532
C01501=1114.916,303.838,-78.052,-177.847,10.495,149.532
C01502=1114.920,303.590,-78.020,-177.850,10.493,149.532
C01503=1114.924,303.341,-77.987,-177.854,10.491,149.532
C01504=1114.929,303.094,-77.956,-177.857,10.488,149.532
C01505=1114.932,302.846,-77.924,-177.860,10.485,149.533
C01506=1114.937,302.597,-77.892,-177.862,10.483,149.533
C01507=1114.941,302.349,-77.860,-177.866,10.481,149.533
C01508=1114.945,302.102,-77.828,-177.869,10.478,149.533
C01509=1114.949,301.854,-77.796,-177.872,10.476,149.533
C01510=1114.953,301.606,-77.764,-177.875,10.473,149.533
C01511=1114.957,301.358,-77.733,-177.878,10.470,149.534
C01512=1114.961,301.110,-77.701,-177.881,10.468,149.534
C01513=1114.966,300.862,-77.668,-177.884,10.465,149.534
C01514=1114.970,300.615,-77.637,-177.887,10.463,149.534
C01515=1114.974,300.367,-77.605,-177.891,10.460,149.534
C01516=1114.977,300.119,-77.573,-177.893,10.458,149.534
C01517=1114.982,299.871,-77.541,-177.896,10.456,149.535
C01518=1114.986,299.623,-77.509,-177.899,10.453,149.535
C01519=1114.990,299.374,-77.478,-177.903,10.450,149.535
C01520=1114.994,299.127,-77.447,-177.905,10.448,149.535
C01521=1114.998,298.879,-77.415,-177.909,10.445,149.535
C01522=1115.002,298.630,-77.382,-177.912,10.443,149.535
C01523=1115.007,298.383,-77.351,-177.915,10.440,149.536
C01524=1115.010,298.135,-77.319,-177.918,10.437,149.536
C01525=1115.014,297.886,-77.288,-177.921,10.435,149.536
C01526=1115.019,297.639,-77.256,-177.924,10.433,149.536
C01527=1115.022,297.391,-77.224,-177.927,10.430,149.536
C01528=1115.027,297.144,-77.193,-177.930,10.428,149.537
C01529=1115.031,296.895,-77.162,-177.933,10.425,149.537
C01530=1115.035,296.647,-77.129,-177.936,10.422,149.537
C01531=1115.040,296.399,-77.098,-177.939,10.420,149.537
C01532=1115.044,296.151,-77.067,-177.942,10.417,149.537
C01533=1115.048,295.903,-77.035,-177.945,10.415,149.537
C01534=1115.052,295.655,-77.003,-177.949,10.412,149.538
C01535=1115.056,295.407,-76.973,-177.951,10.410,149.538
C01536=1115.060,295.159,-76.941,-177.954,10.408,149.538
C01537=1115.064,294.947,-76.914,-177.957,10.405,149.538
C01538=1115.067,294.734,-76.888,-177.960,10.403,149.538
C01539=1115.071,294.522,-76.861,-177.962,10.401,149.538
C01540=1115.074,294.309,-76.833,-177.965,10.399,149.539
C01541=1115.077,294.096,-76.806,-177.968,10.397,149.539
C01542=1115.081,293.883,-76.780,-177.970,10.395,149.539
C01543=1115.084,293.671,-76.753,-177.973,10.392,149.539
C01544=1115.088,293.458,-76.725,-177.975,10.390,149.539
C01545=1115.093,293.210,-76.695,-177.978,10.387,149.539
C01546=1115.096,292.962,-76.663,-177.982,10.385,149.540
C01547=1115.101,292.714,-76.632,-177.985,10.382,149.540
C01548=1115.104,292.466,-76.601,-177.988,10.380,149.540
C01549=1115.108,292.219,-76.570,-177.991,10.377,149.540
C01550=1115.112,291.970,-76.538,-177.994,10.375,149.540
C01551=1115.117,291.723,-76.507,-177.997,10.373,149.540
C01552=1115.121,291.474,-76.476,-178.000,10.370,149.541
C01553=1115.125,291.227,-76.445,-178.003,10.367,149.541
C01554=1115.129,290.978,-76.414,-178.006,10.365,149.541
C01555=1115.133,290.731,-76.382,-178.009,10.362,149.541
C01556=1115.137,290.482,-76.351,-178.012,10.359,149.541
C01557=1115.141,290.234,-76.321,-178.015,10.357,149.541
C01558=1115.145,289.986,-76.289,-178.018,10.354,149.542
C01559=1115.150,289.738,-76.258,-178.021,10.353,149.542
C01560=1115.154,289.490,-76.227,-178.024,10.350,149.542
C01561=1115.158,289.242,-76.196,-178.027,10.347,149.542
C01562=1115.162,288.994,-76.165,-178.030,10.345,149.542
C01563=1115.166,288.746,-76.134,-178.034,10.342,149.543
C01564=1115.170,288.498,-76.104,-178.037,10.339,149.543
C01565=1115.174,288.250,-76.072,-178.039,10.337,149.543
C01566=1115.179,288.002,-76.041,-178.043,10.334,149.543
C01567=1115.183,287.753,-76.010,-178.046,10.331,149.543
C01568=1115.187,287.506,-75.980,-178.048,10.330,149.543
C01569=1115.191,287.258,-75.949,-178.051,10.327,149.543
C01570=1115.195,287.010,-75.917,-178.055,10.325,149.544
C01571=1115.200,286.762,-75.886,-178.058,10.322,149.544
C01572=1115.203,286.513,-75.856,-178.061,10.319,149.544
C01573=1115.207,286.265,-75.825,-178.064,10.317,149.544
C01574=1115.212,286.017,-75.794,-178.067,10.314,149.544
C01575=1115.215,285.769,-75.764,-178.070,10.312,149.545
C01576=1115.220,285.521,-75.733,-178.073,10.309,149.545
C01577=1115.225,285.273,-75.702,-178.076,10.307,149.545
C01578=1115.228,285.025,-75.672,-178.079,10.304,149.545
C01579=1115.232,284.777,-75.641,-178.082,10.302,149.545
C01580=1115.237,284.529,-75.610,-178.085,10.299,149.545
C01581=1115.240,284.281,-75.580,-178.088,10.296,149.546
C01582=1115.245,284.033,-75.549,-178.091,10.294,149.546
C01583=1115.250,283.785,-75.518,-178.094,10.291,149.546
C01584=1115.253,283.536,-75.488,-178.098,10.289,149.546
C01585=1115.257,283.288,-75.457,-178.101,10.286,149.546
C01586=1115.262,283.040,-75.426,-178.103,10.284,149.546
C01587=1115.265,282.792,-75.396,-178.106,10.282,149.547
C01588=1115.270,282.544,-75.365,-178.109,10.279,149.547
C01589=1115.274,282.296,-75.335,-178.112,10.276,149.547
C01590=1115.278,282.048,-75.304,-178.115,10.274,149.547
C01591=1115.282,281.800,-75.273,-178.118,10.271,149.547
C01592=1115.286,281.552,-75.243,-178.122,10.269,149.548
C01593=1115.290,281.339,-75.216,-178.124,10.267,149.548
C01594=1115.294,281.126,-75.190,-178.127,10.264,149.548
C01595=1115.297,280.913,-75.164,-178.130,10.262,149.548
C01596=1115.301,280.701,-75.138,-178.133,10.259,149.548
C01597=1115.305,280.488,-75.112,-178.135,10.257,149.548
C01598=1115.308,280.275,-75.086,-178.138,10.255,149.548
C01599=1115.312,280.062,-75.060,-178.141,10.253,149.549
C01600=1115.315,279.850,-75.034,-178.143,10.251,149.549
C01601=1115.319,279.602,-75.004,-178.146,10.247,149.549
C01602=1115.324,279.354,-74.973,-178.150,10.245,149.549
C01603=1115.328,279.106,-74.944,-178.153,10.242,149.549
C01604=1115.332,278.857,-74.912,-178.156,10.240,149.549
C01605=1115.336,278.609,-74.882,-178.159,10.237,149.550
C01606=1115.341,278.361,-74.852,-178.162,10.234,149.550
C01607=1115.345,278.113,-74.822,-178.165,10.232,149.550
C01608=1115.349,277.865,-74.791,-178.168,10.229,149.550
C01609=1115.353,277.616,-74.761,-178.171,10.226,149.550
C01610=1115.357,277.369,-74.731,-178.174,10.224,149.550
C01611=1115.361,277.121,-74.701,-178.177,10.221,149.551
C01612=1115.365,276.872,-74.671,-178.180,10.218,149.551
C01613=1115.369,276.625,-74.641,-178.183,10.216,149.551
C01614=1115.374,276.375,-74.611,-178.186,10.214,149.551
C01615=1115.378,276.128,-74.580,-178.189,10.211,149.551
C01616=1115.382,275.879,-74.550,-178.192,10.209,149.551
C01617=1115.386,275.632,-74.520,-178.195,10.206,149.551
C01618=1115.391,275.383,-74.491,-178.198,10.203,149.551
C01619=1115.394,275.136,-74.461,-178.201,10.200,149.552
C01620=1115.399,274.887,-74.430,-178.204,10.197,149.552
C01621=1115.403,274.639,-74.400,-178.207,10.195,149.552
C01622=1115.407,274.390,-74.370,-178.210,10.192,149.552
C01623=1115.411,274.143,-74.340,-178.213,10.190,149.552
C01624=1115.416,273.894,-74.310,-178.216,10.187,149.552
C01625=1115.419,273.647,-74.280,-178.219,10.184,149.552
C01626=1115.424,273.398,-74.251,-178.222,10.181,149.552
C01627=1115.429,273.150,-74.221,-178.224,10.179,149.553
C01628=1115.432,272.902,-74.190,-178.227,10.177,149.553
C01629=1115.437,272.654,-74.161,-178.230,10.174,149.553
C01630=1115.441,272.406,-74.131,-178.233,10.171,149.553
C01631=1115.445,272.157,-74.100,-178.236,10.169,149.553
C01632=1115.449,271.909,-74.071,-178.239,10.166,149.553
C01633=1115.453,271.660,-74.041,-178.242,10.163,149.553
C01634=1115.457,271.413,-74.011,-178.244,10.161,149.553
C01635=1115.461,271.164,-73.982,-178.247,10.158,149.554
C01636=1115.466,270.916,-73.952,-178.250,10.156,149.554
C01637=1115.470,270.668,-73.922,-178.253,10.153,149.554
C01638=1115.474,270.420,-73.892,-178.256,10.150,149.554
C01639=1115.478,270.172,-73.863,-178.259,10.147,149.554
C01640=1115.483,269.923,-73.833,-178.261,10.145,149.554
C01641=1115.487,269.675,-73.804,-178.264,10.143,149.554
C01642=1115.491,269.427,-73.774,-178.267,10.140,149.554
C01643=1115.496,269.179,-73.744,-178.270,10.137,149.554
C01644=1115.500,268.931,-73.714,-178.272,10.135,149.554
C01645=1115.504,268.682,-73.685,-178.275,10.132,149.555
C01646=1115.508,268.434,-73.655,-178.278,10.130,149.555
C01647=1115.512,268.186,-73.626,-178.281,10.127,149.555
C01648=1115.516,267.938,-73.596,-178.284,10.125,149.555
C01649=1115.520,267.726,-73.571,-178.286,10.122,149.555
C01650=1115.524,267.512,-73.546,-178.289,10.120,149.555
C01651=1115.527,267.299,-73.520,-178.291,10.118,149.555
C01652=1115.531,267.087,-73.495,-178.293,10.116,149.555
C01653=1115.535,266.873,-73.470,-178.295,10.114,149.555
C01654=1115.538,266.660,-73.444,-178.298,10.112,149.555
C01655=1115.542,266.448,-73.419,-178.300,10.110,149.556
C01656=1115.546,266.234,-73.394,-178.303,10.107,149.556
C01657=1115.550,265.986,-73.364,-178.305,10.105,149.556
C01658=1115.554,265.738,-73.335,-178.308,10.102,149.556
C01659=1115.558,265.489,-73.305,-178.311,10.100,149.556
C01660=1115.563,265.241,-73.276,-178.313,10.098,149.556
C01661=1115.567,264.993,-73.247,-178.316,10.095,149.556
C01662=1115.572,264.745,-73.217,-178.319,10.093,149.556
C01663=1115.576,264.497,-73.188,-178.321,10.090,149.556
C01664=1115.580,264.249,-73.159,-178.325,10.088,149.557
C01665=1115.584,264.001,-73.129,-178.328,10.085,149.557
C01666=1115.588,263.752,-73.100,-178.331,10.081,149.557
C01667=1115.592,263.504,-73.070,-178.335,10.079,149.557
C01668=1115.596,263.256,-73.041,-178.338,10.076,149.557
C01669=1115.600,263.007,-73.013,-178.341,10.073,149.557
C01670=1115.605,262.760,-72.984,-178.344,10.071,149.558
C01671=1115.609,262.511,-72.954,-178.348,10.067,149.558
C01672=1115.613,262.263,-72.925,-178.350,10.065,149.558
C01673=1115.618,262.015,-72.895,-178.353,10.062,149.558
C01674=1115.622,261.766,-72.866,-178.356,10.059,149.558
C01675=1115.626,261.518,-72.837,-178.359,10.056,149.558
C01676=1115.630,261.270,-72.808,-178.363,10.054,149.559
C01677=1115.635,261.022,-72.779,-178.366,10.051,149.559
C01678=1115.639,260.773,-72.750,-178.369,10.049,149.559
C01679=1115.643,260.525,-72.721,-178.372,10.045,149.559
C01680=1115.647,260.277,-72.691,-178.375,10.042,149.559
C01681=1115.652,260.028,-72.663,-178.378,10.039,149.559
C01682=1115.656,259.781,-72.634,-178.381,10.037,149.559
C01683=1115.660,259.532,-72.605,-178.384,10.034,149.559
C01684=1115.665,259.283,-72.576,-178.387,10.031,149.559
C01685=1115.669,259.035,-72.547,-178.389,10.028,149.559
C01686=1115.672,258.787,-72.518,-178.392,10.025,149.559
C01687=1115.677,258.539,-72.489,-178.395,10.023,149.560
C01688=1115.682,258.291,-72.460,-178.398,10.020,149.560
C01689=1115.686,258.042,-72.431,-178.401,10.017,149.560
C01690=1115.689,257.794,-72.402,-178.404,10.014,149.560
C01691=1115.695,257.546,-72.374,-178.407,10.012,149.560
C01692=1115.699,257.297,-72.344,-178.409,10.008,149.560
C01693=1115.702,257.049,-72.316,-178.412,10.006,149.560
C01694=1115.707,256.801,-72.287,-178.415,10.003,149.560
C01695=1115.712,256.552,-72.258,-178.418,10.000,149.560
C01696=1115.715,256.304,-72.230,-178.420,9.998,149.560
C01697=1115.720,256.056,-72.201,-178.423,9.995,149.560
C01698=1115.724,255.808,-72.172,-178.425,9.993,149.560
C01699=1115.728,255.559,-72.144,-178.426,9.991,149.560
C01700=1115.733,255.311,-72.115,-178.428,9.989,149.560
C01701=1115.737,255.062,-72.085,-178.429,9.987,149.560
C01702=1115.741,254.814,-72.058,-178.431,9.985,149.560
C01703=1115.745,254.566,-72.028,-178.433,9.983,149.560
C01704=1115.749,254.318,-72.000,-178.435,9.981,149.560
C01705=1115.753,254.105,-71.975,-178.437,9.979,149.560
C01706=1115.757,253.891,-71.950,-178.438,9.978,149.560
C01707=1115.761,253.678,-71.927,-178.440,9.976,149.560
C01708=1115.765,253.466,-71.902,-178.443,9.974,149.560
C01709=1115.768,253.253,-71.877,-178.444,9.972,149.560
C01710=1115.772,253.040,-71.852,-178.446,9.970,149.560
C01711=1115.776,252.826,-71.828,-178.449,9.968,149.560
C01712=1115.779,252.613,-71.804,-178.451,9.966,149.561
C01713=1115.784,252.365,-71.775,-178.454,9.963,149.561
C01714=1115.788,252.117,-71.746,-178.457,9.962,149.561
C01715=1115.792,251.868,-71.718,-178.459,9.959,149.561
C01716=1115.796,251.620,-71.690,-178.462,9.956,149.561
C01717=1115.801,251.372,-71.660,-178.466,9.954,149.562
C01718=1115.804,251.124,-71.632,-178.469,9.951,149.562
C01719=1115.809,250.875,-71.604,-178.472,9.949,149.562
C01720=1115.813,250.627,-71.576,-178.476,9.945,149.562
C01721=1115.818,250.378,-71.547,-178.479,9.943,149.562
C01722=1115.821,250.130,-71.518,-178.483,9.940,149.563
C01723=1115.826,249.882,-71.490,-178.487,9.936,149.563
C01724=1115.830,249.633,-71.462,-178.491,9.933,149.563
C01725=1115.835,249.385,-71.433,-178.495,9.930,149.563
C01726=1115.839,249.137,-71.405,-178.499,9.927,149.564
C01727=1115.843,248.889,-71.377,-178.502,9.923,149.564
C01728=1115.848,248.640,-71.349,-178.506,9.920,149.564
C01729=1115.851,248.391,-71.320,-178.511,9.916,149.564
C01730=1115.856,248.143,-71.292,-178.515,9.913,149.565
C01731=1115.860,247.894,-71.264,-178.519,9.908,149.565
C01732=1115.865,247.647,-71.236,-178.524,9.904,149.565
C01733=1115.869,247.398,-71.207,-178.527,9.901,149.565
C01734=1115.873,247.150,-71.180,-178.529,9.899,149.565
C01735=1115.877,246.901,-71.152,-178.531,9.896,149.565
C01736=1115.882,246.653,-71.123,-178.533,9.893,149.565
C01737=1115.886,246.404,-71.095,-178.535,9.891,149.565
C01738=1115.890,246.157,-71.067,-178.537,9.888,149.565
C01739=1115.895,245.908,-71.039,-178.540,9.885,149.565
C01740=1115.899,245.660,-71.011,-178.542,9.883,149.565
C01741=1115.903,245.411,-70.983,-178.544,9.881,149.564
C01742=1115.908,245.162,-70.955,-178.545,9.878,149.564
C01743=1115.912,244.914,-70.927,-178.548,9.875,149.564
C01744=1115.916,244.666,-70.899,-178.550,9.873,149.564
C01745=1115.920,244.417,-70.871,-178.552,9.871,149.564
C01746=1115.925,244.169,-70.843,-178.555,9.868,149.564
C01747=1115.929,243.921,-70.814,-178.557,9.866,149.564
C01748=1115.934,243.672,-70.787,-178.559,9.863,149.564
C01749=1115.937,243.424,-70.759,-178.561,9.860,149.564
C01750=1115.943,243.175,-70.731,-178.563,9.858,149.564
C01751=1115.947,242.928,-70.703,-178.566,9.855,149.564
C01752=1115.951,242.678,-70.676,-178.568,9.853,149.564
C01753=1115.955,242.430,-70.648,-178.570,9.851,149.564
C01754=1115.959,242.182,-70.620,-178.573,9.848,149.564
C01755=1115.964,241.934,-70.591,-178.575,9.846,149.564
C01756=1115.968,241.684,-70.564,-178.578,9.843,149.564
C01757=1115.973,241.437,-70.536,-178.580,9.840,149.564
C01758=1115.977,241.189,-70.508,-178.583,9.838,149.565
C01759=1115.981,240.940,-70.481,-178.585,9.835,149.564
C01760=1115.985,240.692,-70.453,-178.588,9.833,149.565
C01761=1115.990,240.478,-70.429,-178.590,9.831,149.565
C01762=1115.993,240.265,-70.405,-178.592,9.828,149.565
C01763=1115.997,240.052,-70.382,-178.594,9.826,149.565
C01764=1116.000,239.839,-70.357,-178.596,9.824,149.565
C01765=1116.004,239.626,-70.334,-178.598,9.822,149.565
C01766=1116.008,239.412,-70.309,-178.600,9.820,149.565
C01767=1116.011,239.199,-70.286,-178.602,9.818,149.565
C01768=1116.015,238.986,-70.262,-178.605,9.816,149.565
C01769=1116.019,238.738,-70.235,-178.607,9.813,149.565
C01770=1116.024,238.489,-70.207,-178.610,9.811,149.565
C01771=1116.028,238.241,-70.179,-178.613,9.808,149.565
C01772=1116.033,237.993,-70.152,-178.616,9.805,149.565
C01773=1116.036,237.744,-70.124,-178.617,9.803,149.565
C01774=1116.041,237.496,-70.097,-178.620,9.800,149.565
C01775=1116.045,237.248,-70.069,-178.623,9.797,149.566
C01776=1116.049,236.998,-70.042,-178.626,9.795,149.566
C01777=1116.054,236.751,-70.014,-178.629,9.793,149.566
C01778=1116.058,236.502,-69.987,-178.631,9.790,149.566
C01779=1116.062,236.253,-69.960,-178.634,9.787,149.566
C01780=1116.067,236.005,-69.932,-178.637,9.784,149.566
C01781=1116.071,235.757,-69.905,-178.639,9.782,149.566
C01782=1116.075,235.508,-69.877,-178.642,9.779,149.566
C01783=1116.080,235.259,-69.850,-178.645,9.777,149.566
C01784=1116.084,235.011,-69.823,-178.648,9.773,149.566
C01785=1116.089,234.763,-69.795,-178.651,9.771,149.566
